            'The directory service has exhausted the pool of relative identifiers.';
    Win32ErrorCodes.ERROR_DS_INCORRECT_ROLE_OWNER:
        Win32ErrorCodeDescription := 'The requested operation could not be performed because the directory service is not the master for that type of operation.';
    Win32ErrorCodes.ERROR_DS_RIDMGR_INIT_ERROR:
        Win32ErrorCodeDescription := 'The directory service was unable to initialize the subsystem that allocates relative identifiers.';
    Win32ErrorCodes.ERROR_DS_OBJ_CLASS_VIOLATION:
        Win32ErrorCodeDescription := 'The requested operation did not satisfy one or more constraints associated with the class of the object.';
    Win32ErrorCodes.ERROR_DS_CANT_ON_NON_LEAF:
        Win32ErrorCodeDescription :=
            'The directory service can perform the requested operation only on a leaf object.';
    Win32ErrorCodes.ERROR_DS_CANT_ON_RDN:
        Win32ErrorCodeDescription := 'The directory service cannot perform the requested operation on the RDN attribute of an object.';
    Win32ErrorCodes.ERROR_DS_CANT_MOD_OBJ_CLASS:
        Win32ErrorCodeDescription :=
            'The directory service detected an attempt to modify the object class of an object.';
    Win32ErrorCodes.ERROR_DS_CROSS_DOM_MOVE_ERROR:
        Win32ErrorCodeDescription :=
            'The requested cross-domain move operation could not be performed.';
    Win32ErrorCodes.ERROR_DS_GC_NOT_AVAILABLE:
        Win32ErrorCodeDescription := 'Unable to contact the global catalog server.';
    Win32ErrorCodes.ERROR_SHARED_POLICY:
        Win32ErrorCodeDescription :=
            'The policy object is shared and can only be modified at the root.';
    Win32ErrorCodes.ERROR_POLICY_OBJECT_NOT_FOUND:
        Win32ErrorCodeDescription := 'The policy object does not exist.';
    Win32ErrorCodes.ERROR_POLICY_ONLY_IN_DS:
        Win32ErrorCodeDescription :=
            'The requested policy information is only in the directory service.';
    Win32ErrorCodes.ERROR_PROMOTION_ACTIVE:
        Win32ErrorCodeDescription := 'A domain controller promotion is currently active.';
    Win32ErrorCodes.ERROR_NO_PROMOTION_ACTIVE:
        Win32ErrorCodeDescription := 'A domain controller promotion is not currently active';
    Win32ErrorCodes.ERROR_DS_OPERATIONS_ERROR:
        Win32ErrorCodeDescription := 'An operations error occurred.';
    Win32ErrorCodes.ERROR_DS_PROTOCOL_ERROR:
        Win32ErrorCodeDescription := 'A protocol error occurred.';
    Win32ErrorCodes.ERROR_DS_TIMELIMIT_EXCEEDED:
        Win32ErrorCodeDescription := 'The time limit for this request was exceeded.';
    Win32ErrorCodes.ERROR_DS_SIZELIMIT_EXCEEDED:
        Win32ErrorCodeDescription := 'The size limit for this request was exceeded.';
    Win32ErrorCodes.ERROR_DS_ADMIN_LIMIT_EXCEEDED:
        Win32ErrorCodeDescription := 'The administrative limit for this request was exceeded.';
    Win32ErrorCodes.ERROR_DS_COMPARE_FALSE:
        Win32ErrorCodeDescription := 'The compare response was false.';
    Win32ErrorCodes.ERROR_DS_COMPARE_TRUE:
        Win32ErrorCodeDescription := 'The compare response was true.';
    Win32ErrorCodes.ERROR_DS_AUTH_METHOD_NOT_SUPPORTED:
        Win32ErrorCodeDescription :=
            'The requested authentication method is not supported by the server.';
    Win32ErrorCodes.ERROR_DS_STRONG_AUTH_REQUIRED:
        Win32ErrorCodeDescription :=
            'A more secure authentication method is required for this server.';
    Win32ErrorCodes.ERROR_DS_INAPPROPRIATE_AUTH:
        Win32ErrorCodeDescription := 'Inappropriate authentication.';
    Win32ErrorCodes.ERROR_DS_AUTH_UNKNOWN:
        Win32ErrorCodeDescription := 'The authentication mechanism is unknown.';
    Win32ErrorCodes.ERROR_DS_REFERRAL:
        Win32ErrorCodeDescription := 'A referral was returned from the server.';
    Win32ErrorCodes.ERROR_DS_UNAVAILABLE_CRIT_EXTENSION:
        Win32ErrorCodeDescription :=
            'The server does not support the requested critical extension.';
    Win32ErrorCodes.ERROR_DS_CONFIDENTIALITY_REQUIRED:
        Win32ErrorCodeDescription := 'This request requires a secure connection.';
    Win32ErrorCodes.ERROR_DS_INAPPROPRIATE_MATCHING:
        Win32ErrorCodeDescription := 'Inappropriate matching.';
    Win32ErrorCodes.ERROR_DS_CONSTRAINT_VIOLATION:
        Win32ErrorCodeDescription := 'A constraint violation occurred.';
    Win32ErrorCodes.ERROR_DS_NO_SUCH_OBJECT:
        Win32ErrorCodeDescription := 'There is no such object on the server.';
    Win32ErrorCodes.ERROR_DS_ALIAS_PROBLEM:
        Win32ErrorCodeDescription := 'There is an alias problem.';
    Win32ErrorCodes.ERROR_DS_INVALID_DN_SYNTAX:
        Win32ErrorCodeDescription := 'An invalid dn syntax has been specified.';
    Win32ErrorCodes.ERROR_DS_IS_LEAF:
        Win32ErrorCodeDescription := 'The object is a leaf object.';
    Win32ErrorCodes.ERROR_DS_ALIAS_DEREF_PROBLEM:
        Win32ErrorCodeDescription := 'There is an alias dereferencing problem.';
    Win32ErrorCodes.ERROR_DS_UNWILLING_TO_PERFORM:
        Win32ErrorCodeDescription := 'The server is unwilling to process the request.';
    Win32ErrorCodes.ERROR_DS_LOOP_DETECT:
        Win32ErrorCodeDescription := 'A loop has been detected.';
    Win32ErrorCodes.ERROR_DS_NAMING_VIOLATION:
        Win32ErrorCodeDescription := 'There is a naming violation.';
    Win32ErrorCodes.ERROR_DS_OBJECT_RESULTS_TOO_LARGE:
        Win32ErrorCodeDescription := 'The result set is too large.';
    Win32ErrorCodes.ERROR_DS_AFFECTS_MULTIPLE_DSAS:
        Win32ErrorCodeDescription := 'The operation affects multiple DSAs';
    Win32ErrorCodes.ERROR_DS_SERVER_DOWN:
        Win32ErrorCodeDescription := 'The server is not operational.';
    Win32ErrorCodes.ERROR_DS_LOCAL_ERROR:
        Win32ErrorCodeDescription := 'A local error has occurred.';
    Win32ErrorCodes.ERROR_DS_ENCODING_ERROR:
        Win32ErrorCodeDescription := 'An encoding error has occurred.';
    Win32ErrorCodes.ERROR_DS_DECODING_ERROR:
        Win32ErrorCodeDescription := 'A decoding error has occurred.';
    Win32ErrorCodes.ERROR_DS_FILTER_UNKNOWN:
        Win32ErrorCodeDescription := 'The search filter cannot be recognized.';
    Win32ErrorCodes.ERROR_DS_PARAM_ERROR:
        Win32ErrorCodeDescription := 'One or more parameters are illegal.';
    Win32ErrorCodes.ERROR_DS_NOT_SUPPORTED:
        Win32ErrorCodeDescription := 'The specified method is not supported.';
    Win32ErrorCodes.ERROR_DS_NO_RESULTS_RETURNED:
        Win32ErrorCodeDescription := 'No results were returned.';
    Win32ErrorCodes.ERROR_DS_CONTROL_NOT_FOUND:
        Win32ErrorCodeDescription := 'The specified control is not supported by the server.';
    Win32ErrorCodes.ERROR_DS_CLIENT_LOOP:
        Win32ErrorCodeDescription := 'A referral loop was detected by the client.';
    Win32ErrorCodes.ERROR_DS_REFERRAL_LIMIT_EXCEEDED:
        Win32ErrorCodeDescription := 'The preset referral limit was exceeded.';
    Win32ErrorCodes.ERROR_DS_SORT_CONTROL_MISSING:
        Win32ErrorCodeDescription := 'The search requires a SORT control.';
    Win32ErrorCodes.ERROR_DS_OFFSET_RANGE_ERROR:
        Win32ErrorCodeDescription := 'The search results exceed the offset range specified.';
    Win32ErrorCodes.ERROR_DS_ROOT_MUST_BE_NC:
        Win32ErrorCodeDescription := 'The root object must be the head of a naming context. The root object cannot have an instantiated parent.';
    Win32ErrorCodes.ERROR_DS_ADD_REPLICA_INHIBITED:
        Win32ErrorCodeDescription := 'The add replica operation cannot be performed. The naming context must be writable in order to create the replica.';
    Win32ErrorCodes.ERROR_DS_ATT_NOT_DEF_IN_SCHEMA:
        Win32ErrorCodeDescription :=
            'A reference to an attribute that is not defined in the schema occurred.';
    Win32ErrorCodes.ERROR_DS_MAX_OBJ_SIZE_EXCEEDED:
        Win32ErrorCodeDescription := 'The maximum size of an object has been exceeded.';
    Win32ErrorCodes.ERROR_DS_OBJ_STRING_NAME_EXISTS:
        Win32ErrorCodeDescription :=
            'An attempt was made to add an object to the directory with a name that is already in use.';
    Win32ErrorCodes.ERROR_DS_NO_RDN_DEFINED_IN_SCHEMA:
        Win32ErrorCodeDescription := 'An attempt was made to add an object of a class that does not have an RDN defined in the schema.';
    Win32ErrorCodes.ERROR_DS_RDN_DOESNT_MATCH_SCHEMA:
        Win32ErrorCodeDescription := 'An attempt was made to add an object using an RDN that is not the RDN defined in the schema.';
    Win32ErrorCodes.ERROR_DS_NO_REQUESTED_ATTS_FOUND:
        Win32ErrorCodeDescription := 'None of the requested attributes were found on the objects.';
    Win32ErrorCodes.ERROR_DS_USER_BUFFER_TO_SMALL:
        Win32ErrorCodeDescription := 'The user buffer is too small.';
    Win32ErrorCodes.ERROR_DS_ATT_IS_NOT_ON_OBJ:
        Win32ErrorCodeDescription :=
            'The attribute specified in the operation is not present on the object.';
    Win32ErrorCodes.ERROR_DS_ILLEGAL_MOD_OPERATION:
        Win32ErrorCodeDescription :=
            'Illegal modify operation. Some aspect of the modification is not permitted.';
    Win32ErrorCodes.ERROR_DS_OBJ_TOO_LARGE:
        Win32ErrorCodeDescription := 'The specified object is too large.';
    Win32ErrorCodes.ERROR_DS_BAD_INSTANCE_TYPE:
        Win32ErrorCodeDescription := 'The specified instance type is not valid.';
    Win32ErrorCodes.ERROR_DS_MASTERDSA_REQUIRED:
        Win32ErrorCodeDescription := 'The operation must be performed at a master DSA.';
    Win32ErrorCodes.ERROR_DS_OBJECT_CLASS_REQUIRED:
        Win32ErrorCodeDescription := 'The object class attribute must be specified.';
    Win32ErrorCodes.ERROR_DS_MISSING_REQUIRED_ATT:
        Win32ErrorCodeDescription := 'A required attribute is missing.';
    Win32ErrorCodes.ERROR_DS_ATT_NOT_DEF_FOR_CLASS:
        Win32ErrorCodeDescription := 'An attempt was made to modify an object to include an attribute that is not legal for its class';
    Win32ErrorCodes.ERROR_DS_ATT_ALREADY_EXISTS:
        Win32ErrorCodeDescription := 'The specified attribute is already present on the object.';
    Win32ErrorCodes.ERROR_DS_CANT_ADD_ATT_VALUES:
        Win32ErrorCodeDescription := 'The specified attribute is not present, or has no values.';
    Win32ErrorCodes.ERROR_DS_SINGLE_VALUE_CONSTRAINT:
        Win32ErrorCodeDescription :=
            'Multiple values were specified for an attribute that can have only one value.';
    Win32ErrorCodes.ERROR_DS_RANGE_CONSTRAINT:
        Win32ErrorCodeDescription :=
            'A value for the attribute was not in the acceptable range of values.';
    Win32ErrorCodes.ERROR_DS_ATT_VAL_ALREADY_EXISTS:
        Win32ErrorCodeDescription := 'The specified value already exists.';
    Win32ErrorCodes.ERROR_DS_CANT_REM_MISSING_ATT:
        Win32ErrorCodeDescription :=
            'The attribute cannot be removed because it is not present on the object.';
    Win32ErrorCodes.ERROR_DS_CANT_REM_MISSING_ATT_VAL:
        Win32ErrorCodeDescription :=
            'The attribute value cannot be removed because it is not present on the object.';
    Win32ErrorCodes.ERROR_DS_ROOT_CANT_BE_SUBREF:
        Win32ErrorCodeDescription := 'The specified root object cannot be a subref.';
    Win32ErrorCodes.ERROR_DS_NO_CHAINING:
        Win32ErrorCodeDescription := 'Chaining is not permitted.';
    Win32ErrorCodes.ERROR_DS_NO_CHAINED_EVAL:
        Win32ErrorCodeDescription := 'Chained evaluation is not permitted.';
    Win32ErrorCodes.ERROR_DS_NO_PARENT_OBJECT:
        Win32ErrorCodeDescription := 'The operation could not be performed because the objects parent is either uninstantiated or deleted.';
    Win32ErrorCodes.ERROR_DS_PARENT_IS_AN_ALIAS:
        Win32ErrorCodeDescription :=
            'Having a parent that is an alias is not permitted. Aliases are leaf objects.';
    Win32ErrorCodes.ERROR_DS_CANT_MIX_MASTER_AND_REPS:
        Win32ErrorCodeDescription :=
            'The object and parent must be of the same type, either both masters or both replicas.';
    Win32ErrorCodes.ERROR_DS_CHILDREN_EXIST:
        Win32ErrorCodeDescription := 'The operation cannot be performed because child objects exist. This operation can only be performed on a leaf object.';
    Win32ErrorCodes.ERROR_DS_OBJ_NOT_FOUND:
        Win32ErrorCodeDescription := 'Directory object not found.';
    Win32ErrorCodes.ERROR_DS_ALIASED_OBJ_MISSING:
        Win32ErrorCodeDescription := 'The aliased object is missing.';
    Win32ErrorCodes.ERROR_DS_BAD_NAME_SYNTAX:
        Win32ErrorCodeDescription := 'The object name has bad syntax.';
    Win32ErrorCodes.ERROR_DS_ALIAS_POINTS_TO_ALIAS:
        Win32ErrorCodeDescription := 'It is not permitted for an alias to refer to another alias.';
    Win32ErrorCodes.ERROR_DS_CANT_DEREF_ALIAS:
        Win32ErrorCodeDescription := 'The alias cannot be dereferenced.';
    Win32ErrorCodes.ERROR_DS_OUT_OF_SCOPE:
        Win32ErrorCodeDescription := 'The operation is out of scope.';
    Win32ErrorCodes.ERROR_DS_OBJECT_BEING_REMOVED:
        Win32ErrorCodeDescription :=
            'The operation cannot continue because the object is in the process of being removed.';
    Win32ErrorCodes.ERROR_DS_CANT_DELETE_DSA_OBJ:
        Win32ErrorCodeDescription := 'The DSA object cannot be deleted.';
    Win32ErrorCodes.ERROR_DS_GENERIC_ERROR:
        Win32ErrorCodeDescription := 'A directory service error has occurred.';
    Win32ErrorCodes.ERROR_DS_DSA_MUST_BE_INT_MASTER:
        Win32ErrorCodeDescription :=
            'The operation can only be performed on an internal master DSA object.';
    Win32ErrorCodes.ERROR_DS_CLASS_NOT_DSA:
        Win32ErrorCodeDescription := 'The object must be of class DSA.';
    Win32ErrorCodes.ERROR_DS_INSUFF_ACCESS_RIGHTS:
        Win32ErrorCodeDescription := 'Insufficient access rights to perform the operation.';
    Win32ErrorCodes.ERROR_DS_ILLEGAL_SUPERIOR:
        Win32ErrorCodeDescription :=
            'The object cannot be added because the parent is not on the list of possible superiors.';
    Win32ErrorCodes.ERROR_DS_ATTRIBUTE_OWNED_BY_SAM:
        Win32ErrorCodeDescription := 'Access to the attribute is not permitted because the attribute is owned by the Security Accounts Manager (SAM).';
    Win32ErrorCodes.ERROR_DS_NAME_TOO_MANY_PARTS:
        Win32ErrorCodeDescription := 'The name has too many parts.';
    Win32ErrorCodes.ERROR_DS_NAME_TOO_LONG:
        Win32ErrorCodeDescription := 'The name is too long.';
    Win32ErrorCodes.ERROR_DS_NAME_VALUE_TOO_LONG:
        Win32ErrorCodeDescription := 'The name value is too long.';
    Win32ErrorCodes.ERROR_DS_NAME_UNPARSEABLE:
        Win32ErrorCodeDescription := 'The directory service encountered an error parsing a name.';
    Win32ErrorCodes.ERROR_DS_NAME_TYPE_UNKNOWN:
        Win32ErrorCodeDescription :=
            'The directory service cannot get the attribute type for a name.';
    Win32ErrorCodes.ERROR_DS_NOT_AN_OBJECT:
        Win32ErrorCodeDescription :=
            'The name does not identify an object; the name identifies a phantom.';
    Win32ErrorCodes.ERROR_DS_SEC_DESC_TOO_SHORT:
        Win32ErrorCodeDescription := 'The security descriptor is too short.';
    Win32ErrorCodes.ERROR_DS_SEC_DESC_INVALID:
        Win32ErrorCodeDescription := 'The security descriptor is invalid.';
    Win32ErrorCodes.ERROR_DS_NO_DELETED_NAME:
        Win32ErrorCodeDescription := 'Failed to create name for deleted object.';
    Win32ErrorCodes.ERROR_DS_SUBREF_MUST_HAVE_PARENT:
        Win32ErrorCodeDescription := 'The parent of a new subref must exist.';
    Win32ErrorCodes.ERROR_DS_NCNAME_MUST_BE_NC:
        Win32ErrorCodeDescription := 'The object must be a naming context.';
    Win32ErrorCodes.ERROR_DS_CANT_ADD_SYSTEM_ONLY:
        Win32ErrorCodeDescription :=
            'It is not permitted to add an attribute which is owned by the system.';
    Win32ErrorCodes.ERROR_DS_CLASS_MUST_BE_CONCRETE:
        Win32ErrorCodeDescription :=
            'The class of the object must be structural; you cannot instantiate an abstract class.';
    Win32ErrorCodes.ERROR_DS_INVALID_DMD:
        Win32ErrorCodeDescription := 'The schema object could not be found.';
    Win32ErrorCodes.ERROR_DS_OBJ_GUID_EXISTS:
        Win32ErrorCodeDescription :=
            'A local object with this GUID (dead or alive) already exists.';
    Win32ErrorCodes.ERROR_DS_NOT_ON_BACKLINK:
        Win32ErrorCodeDescription := 'The operation cannot be performed on a back link.';
    Win32ErrorCodes.ERROR_DS_NO_CROSSREF_FOR_NC:
        Win32ErrorCodeDescription :=
            'The cross reference for the specified naming context could not be found.';
    Win32ErrorCodes.ERROR_DS_SHUTTING_DOWN:
        Win32ErrorCodeDescription :=
            'The operation could not be performed because the directory service is shutting down.';
    Win32ErrorCodes.ERROR_DS_UNKNOWN_OPERATION:
        Win32ErrorCodeDescription := 'The directory service request is invalid.';
    Win32ErrorCodes.ERROR_DS_INVALID_ROLE_OWNER:
        Win32ErrorCodeDescription := 'The role owner attribute could not be read.';
    Win32ErrorCodes.ERROR_DS_COULDNT_CONTACT_FSMO:
        Win32ErrorCodeDescription :=
            'The requested FSMO operation failed. The current FSMO holder could not be reached.';
    Win32ErrorCodes.ERROR_DS_CROSS_NC_DN_RENAME:
        Win32ErrorCodeDescription :=
            'Modification of a DN across a naming context is not permitted.';
    Win32ErrorCodes.ERROR_DS_CANT_MOD_SYSTEM_ONLY:
        Win32ErrorCodeDescription :=
            'The attribute cannot be modified because it is owned by the system.';
    Win32ErrorCodes.ERROR_DS_REPLICATOR_ONLY:
        Win32ErrorCodeDescription := 'Only the replicator can perform this function.';
    Win32ErrorCodes.ERROR_DS_OBJ_CLASS_NOT_DEFINED:
        Win32ErrorCodeDescription := 'The specified class is not defined.';
    Win32ErrorCodes.ERROR_DS_OBJ_CLASS_NOT_SUBCLASS:
        Win32ErrorCodeDescription := 'The specified class is not a subclass.';
    Win32ErrorCodes.ERROR_DS_NAME_REFERENCE_INVALID:
        Win32ErrorCodeDescription := 'The name reference is invalid.';
    Win32ErrorCodes.ERROR_DS_CROSS_REF_EXISTS:
        Win32ErrorCodeDescription := 'A cross reference already exists.';
    Win32ErrorCodes.ERROR_DS_CANT_DEL_MASTER_CROSSREF:
        Win32ErrorCodeDescription := 'It is not permitted to delete a master cross reference.';
    Win32ErrorCodes.ERROR_DS_SUBTREE_NOTIFY_NOT_NC_HEAD:
        Win32ErrorCodeDescription := 'Subtree notifications are only supported on NC heads.';
    Win32ErrorCodes.ERROR_DS_NOTIFY_FILTER_TOO_COMPLEX:
        Win32ErrorCodeDescription := 'Notification filter is too complex.';
    Win32ErrorCodes.ERROR_DS_DUP_RDN:
        Win32ErrorCodeDescription := 'Schema update failed: duplicate RDN.';
    Win32ErrorCodes.ERROR_DS_DUP_OID:
        Win32ErrorCodeDescription := 'Schema update failed: duplicate OID';
    Win32ErrorCodes.ERROR_DS_DUP_MAPI_ID:
        Win32ErrorCodeDescription := 'Schema update failed: duplicate MAPI identifier.';
    Win32ErrorCodes.ERROR_DS_DUP_SCHEMA_ID_GUID:
        Win32ErrorCodeDescription := 'Schema update failed: duplicate schema-id GUID.';
    Win32ErrorCodes.ERROR_DS_DUP_LDAP_DISPLAY_NAME:
        Win32ErrorCodeDescription := 'Schema update failed: duplicate LDAP display name.';
    Win32ErrorCodes.ERROR_DS_SEMANTIC_ATT_TEST:
        Win32ErrorCodeDescription := 'Schema update failed: range-lower less than range upper';
    Win32ErrorCodes.ERROR_DS_SYNTAX_MISMATCH:
        Win32ErrorCodeDescription := 'Schema update failed: syntax mismatch';
    Win32ErrorCodes.ERROR_DS_EXISTS_IN_MUST_HAVE:
        Win32ErrorCodeDescription := 'Schema deletion failed: attribute is used in must-contain';
    Win32ErrorCodes.ERROR_DS_EXISTS_IN_MAY_HAVE:
        Win32ErrorCodeDescription := 'Schema deletion failed: attribute is used in may-contain';
    Win32ErrorCodes.ERROR_DS_NONEXISTENT_MAY_HAVE:
        Win32ErrorCodeDescription :=
            'Schema update failed: attribute in may-contain does not exist';
    Win32ErrorCodes.ERROR_DS_NONEXISTENT_MUST_HAVE:
        Win32ErrorCodeDescription :=
            'Schema update failed: attribute in must-contain does not exist';
    Win32ErrorCodes.ERROR_DS_AUX_CLS_TEST_FAIL:
        Win32ErrorCodeDescription :=
            'Schema update failed: class in aux-class list does not exist or is not an auxiliary class';
    Win32ErrorCodes.ERROR_DS_NONEXISTENT_POSS_SUP:
        Win32ErrorCodeDescription :=
            'Schema update failed: class in poss-superiors does not exist';
    Win32ErrorCodes.ERROR_DS_SUB_CLS_TEST_FAIL:
        Win32ErrorCodeDescription := 'Schema update failed: class in subclassof list does not exist or does not satisfy hierarchy rules';
    Win32ErrorCodes.ERROR_DS_BAD_RDN_ATT_ID_SYNTAX:
        Win32ErrorCodeDescription := 'Schema update failed: Rdn-Att-Id has wrong syntax';
    Win32ErrorCodes.ERROR_DS_EXISTS_IN_AUX_CLS:
        Win32ErrorCodeDescription := 'Schema deletion failed: class is used as auxiliary class';
    Win32ErrorCodes.ERROR_DS_EXISTS_IN_SUB_CLS:
        Win32ErrorCodeDescription := 'Schema deletion failed: class is used as sub class';
    Win32ErrorCodes.ERROR_DS_EXISTS_IN_POSS_SUP:
        Win32ErrorCodeDescription := 'Schema deletion failed: class is used as poss superior';
    Win32ErrorCodes.ERROR_DS_RECALCSCHEMA_FAILED:
        Win32ErrorCodeDescription := 'Schema update failed in recalculating validation cache.';
    Win32ErrorCodes.ERROR_DS_TREE_DELETE_NOT_FINISHED:
        Win32ErrorCodeDescription := 'The tree deletion is not finished.';
    Win32ErrorCodes.ERROR_DS_CANT_DELETE:
        Win32ErrorCodeDescription := 'The requested delete operation could not be performed.';
    Win32ErrorCodes.ERROR_DS_ATT_SCHEMA_REQ_ID:
        Win32ErrorCodeDescription :=
            'Cannot read the governs class identifier for the schema record.';
    Win32ErrorCodes.ERROR_DS_BAD_ATT_SCHEMA_SYNTAX:
        Win32ErrorCodeDescription := 'The attribute schema has bad syntax.';
    Win32ErrorCodes.ERROR_DS_CANT_CACHE_ATT:
        Win32ErrorCodeDescription := 'The attribute could not be cached.';
    Win32ErrorCodes.ERROR_DS_CANT_CACHE_CLASS:
        Win32ErrorCodeDescription := 'The class could not be cached.';
    Win32ErrorCodes.ERROR_DS_CANT_REMOVE_ATT_CACHE:
        Win32ErrorCodeDescription := 'The attribute could not be removed from the cache.';
    Win32ErrorCodes.ERROR_DS_CANT_REMOVE_CLASS_CACHE:
        Win32ErrorCodeDescription := 'The class could not be removed from the cache.';
    Win32ErrorCodes.ERROR_DS_CANT_RETRIEVE_DN:
        Win32ErrorCodeDescription := 'The distinguished name attribute could not be read.';
    Win32ErrorCodes.ERROR_DS_MISSING_SUPREF:
        Win32ErrorCodeDescription := 'A required subref is missing.';
    Win32ErrorCodes.ERROR_DS_CANT_RETRIEVE_INSTANCE:
        Win32ErrorCodeDescription := 'The instance type attribute could not be retrieved.';
    Win32ErrorCodes.ERROR_DS_CODE_INCONSISTENCY:
        Win32ErrorCodeDescription := 'An internal error has occurred.';
    Win32ErrorCodes.ERROR_DS_DATABASE_ERROR:
        Win32ErrorCodeDescription := 'A database error has occurred.';
    Win32ErrorCodes.ERROR_DS_GOVERNSID_MISSING:
        Win32ErrorCodeDescription := 'The attribute GOVERNSID is missing.';
    Win32ErrorCodes.ERROR_DS_MISSING_EXPECTED_ATT:
        Win32ErrorCodeDescription := 'An expected attribute is missing.';
    Win32ErrorCodes.ERROR_DS_NCNAME_MISSING_CR_REF:
        Win32ErrorCodeDescription := 'The specified naming context is missing a cross reference.';
    Win32ErrorCodes.ERROR_DS_SECURITY_CHECKING_ERROR:
        Win32ErrorCodeDescription := 'A security checking error has occurred.';
    Win32ErrorCodes.ERROR_DS_SCHEMA_NOT_LOADED:
        Win32ErrorCodeDescription := 'The schema is not loaded.';
    Win32ErrorCodes.ERROR_DS_SCHEMA_ALLOC_FAILED:
        Win32ErrorCodeDescription :=
            'Schema allocation failed. Please check if the machine is running low on memory.';
    Win32ErrorCodes.ERROR_DS_ATT_SCHEMA_REQ_SYNTAX:
        Win32ErrorCodeDescription :=
            'Failed to obtain the required syntax for the attribute schema.';
    Win32ErrorCodes.ERROR_DS_GCVERIFY_ERROR:
        Win32ErrorCodeDescription := 'The global catalog verification failed. The global catalog is not available or does not support the operation. Some part of the directory is currently not available.';
    Win32ErrorCodes.ERROR_DS_DRA_SCHEMA_MISMATCH:
        Win32ErrorCodeDescription := 'The replication operation failed because of a schema mismatch between the servers involved.';
    Win32ErrorCodes.ERROR_DS_CANT_FIND_DSA_OBJ:
        Win32ErrorCodeDescription := 'The DSA object could not be found.';
    Win32ErrorCodes.ERROR_DS_CANT_FIND_EXPECTED_NC:
        Win32ErrorCodeDescription := 'The naming context could not be found.';
    Win32ErrorCodes.ERROR_DS_CANT_FIND_NC_IN_CACHE:
        Win32ErrorCodeDescription := 'The naming context could not be found in the cache.';
    Win32ErrorCodes.ERROR_DS_CANT_RETRIEVE_CHILD:
        Win32ErrorCodeDescription := 'The child object could not be retrieved.';
    Win32ErrorCodes.ERROR_DS_SECURITY_ILLEGAL_MODIFY:
        Win32ErrorCodeDescription := 'The modification was not permitted for security reasons.';
    Win32ErrorCodes.ERROR_DS_CANT_REPLACE_HIDDEN_REC:
        Win32ErrorCodeDescription := 'The operation cannot replace the hidden record.';
    Win32ErrorCodes.ERROR_DS_BAD_HIERARCHY_FILE:
        Win32ErrorCodeDescription := 'The hierarchy file is invalid.';
    Win32ErrorCodes.ERROR_DS_BUILD_HIERARCHY_TABLE_FAILED:
        Win32ErrorCodeDescription := 'The attempt to build the hierarchy table failed.';
    Win32ErrorCodes.ERROR_DS_CONFIG_PARAM_MISSING:
        Win32ErrorCodeDescription :=
            'The directory configuration parameter is missing from the registry.';
    Win32ErrorCodes.ERROR_DS_COUNTING_AB_INDICES_FAILED:
        Win32ErrorCodeDescription := 'The attempt to count the address book indices failed.';
    Win32ErrorCodes.ERROR_DS_HIERARCHY_TABLE_MALLOC_FAILED:
        Win32ErrorCodeDescription := 'The allocation of the hierarchy table failed.';
    Win32ErrorCodes.ERROR_DS_INTERNAL_FAILURE:
        Win32ErrorCodeDescription := 'The directory service encountered an internal failure.';
    Win32ErrorCodes.ERROR_DS_UNKNOWN_ERROR:
        Win32ErrorCodeDescription := 'The directory service encountered an unknown failure.';
    Win32ErrorCodes.ERROR_DS_ROOT_REQUIRES_CLASS_TOP:
        Win32ErrorCodeDescription := 'A root object requires a class of top.';
    Win32ErrorCodes.ERROR_DS_REFUSING_FSMO_ROLES:
        Win32ErrorCodeDescription := 'This directory server is shutting down, and cannot take ownership of new floating single-master operation roles.';
    Win32ErrorCodes.ERROR_DS_MISSING_FSMO_SETTINGS:
        Win32ErrorCodeDescription := 'The directory service is missing mandatory configuration information, and is unable to determine the ownership of floating single-master operation roles.';
    Win32ErrorCodes.ERROR_DS_UNABLE_TO_SURRENDER_ROLES:
        Win32ErrorCodeDescription := 'The directory service was unable to transfer ownership of one or more floating single-master operation roles to other servers.';
    Win32ErrorCodes.ERROR_DS_DRA_GENERIC:
        Win32ErrorCodeDescription := 'The replication operation failed.';
    Win32ErrorCodes.ERROR_DS_DRA_INVALID_PARAMETER:
        Win32ErrorCodeDescription :=
            'An invalid parameter was specified for this replication operation.';
    Win32ErrorCodes.ERROR_DS_DRA_BUSY:
        Win32ErrorCodeDescription :=
            'The directory service is too busy to complete the replication operation at this time.';
    Win32ErrorCodes.ERROR_DS_DRA_BAD_DN:
        Win32ErrorCodeDescription :=
            'The distinguished name specified for this replication operation is invalid.';
    Win32ErrorCodes.ERROR_DS_DRA_BAD_NC:
        Win32ErrorCodeDescription :=
            'The naming context specified for this replication operation is invalid.';
    Win32ErrorCodes.ERROR_DS_DRA_DN_EXISTS:
        Win32ErrorCodeDescription :=
            'The distinguished name specified for this replication operation already exists.';
    Win32ErrorCodes.ERROR_DS_DRA_INTERNAL_ERROR:
        Win32ErrorCodeDescription := 'The replication system encountered an internal error.';
    Win32ErrorCodes.ERROR_DS_DRA_INCONSISTENT_DIT:
        Win32ErrorCodeDescription :=
            'The replication operation encountered a database inconsistency.';
    Win32ErrorCodes.ERROR_DS_DRA_CONNECTION_FAILED:
        Win32ErrorCodeDescription :=
            'The server specified for this replication operation could not be contacted.';
    Win32ErrorCodes.ERROR_DS_DRA_BAD_INSTANCE_TYPE:
        Win32ErrorCodeDescription :=
            'The replication operation encountered an object with an invalid instance type.';
    Win32ErrorCodes.ERROR_DS_DRA_OUT_OF_MEM:
        Win32ErrorCodeDescription := 'The replication operation failed to allocate memory.';
    Win32ErrorCodes.ERROR_DS_DRA_MAIL_PROBLEM:
        Win32ErrorCodeDescription :=
            'The replication operation encountered an error with the mail system.';
    Win32ErrorCodes.ERROR_DS_DRA_REF_ALREADY_EXISTS:
        Win32ErrorCodeDescription :=
            'The replication reference information for the target server already exists.';
    Win32ErrorCodes.ERROR_DS_DRA_REF_NOT_FOUND:
        Win32ErrorCodeDescription :=
            'The replication reference information for the target server does not exist.';
    Win32ErrorCodes.ERROR_DS_DRA_OBJ_IS_REP_SOURCE:
        Win32ErrorCodeDescription :=
            'The naming context cannot be removed because it is replicated to another server.';
    Win32ErrorCodes.ERROR_DS_DRA_DB_ERROR:
        Win32ErrorCodeDescription := 'The replication operation encountered a database error.';
    Win32ErrorCodes.ERROR_DS_DRA_NO_REPLICA:
        Win32ErrorCodeDescription := 'The naming context is in the process of being removed or is not replicated from the specified server.';
    Win32ErrorCodes.ERROR_DS_DRA_ACCESS_DENIED:
        Win32ErrorCodeDescription := 'Replication access was denied.';
    Win32ErrorCodes.ERROR_DS_DRA_NOT_SUPPORTED:
        Win32ErrorCodeDescription :=
            'The requested operation is not supported by this version of the directory service.';
    Win32ErrorCodes.ERROR_DS_DRA_RPC_CANCELLED:
        Win32ErrorCodeDescription := 'The replication remote procedure call was cancelled.';
    Win32ErrorCodes.ERROR_DS_DRA_SOURCE_DISABLED:
        Win32ErrorCodeDescription :=
            'The source server is currently rejecting replication requests.';
    Win32ErrorCodes.ERROR_DS_DRA_SINK_DISABLED:
        Win32ErrorCodeDescription :=
            'The destination server is currently rejecting replication requests.';
    Win32ErrorCodes.ERROR_DS_DRA_NAME_COLLISION:
        Win32ErrorCodeDescription :=
            'The replication operation failed due to a collision of object names.';
    Win32ErrorCodes.ERROR_DS_DRA_SOURCE_REINSTALLED:
        Win32ErrorCodeDescription := 'The replication source has been reinstalled.';
    Win32ErrorCodes.ERROR_DS_DRA_MISSING_PARENT:
        Win32ErrorCodeDescription :=
            'The replication operation failed because a required parent object is missing.';
    Win32ErrorCodes.ERROR_DS_DRA_PREEMPTED:
        Win32ErrorCodeDescription := 'The replication operation was preempted.';
    Win32ErrorCodes.ERROR_DS_DRA_ABANDON_SYNC:
        Win32ErrorCodeDescription :=
            'The replication synchronization attempt was abandoned because of a lack of updates.';
    Win32ErrorCodes.ERROR_DS_DRA_SHUTDOWN:
        Win32ErrorCodeDescription :=
            'The replication operation was terminated because the system is shutting down.';
    Win32ErrorCodes.ERROR_DS_DRA_INCOMPATIBLE_PARTIAL_SET:
        Win32ErrorCodeDescription := 'The replication synchronization attempt failed as the destination partial attribute set is not a subset of source partial attribute set.';
    Win32ErrorCodes.ERROR_DS_DRA_SOURCE_IS_PARTIAL_REPLICA:
        Win32ErrorCodeDescription := 'The replication synchronization attempt failed because a master replica attempted to sync from a partial replica.';
    Win32ErrorCodes.ERROR_DS_DRA_EXTN_CONNECTION_FAILED:
        Win32ErrorCodeDescription := 'The server specified for this replication operation was contacted, but that server was unable to contact an additional server needed to complete the operation.';
    Win32ErrorCodes.ERROR_DS_INSTALL_SCHEMA_MISMATCH:
        Win32ErrorCodeDescription := 'The version of the Active Directory (AD) schema of the source forest is not compatible with the version of AD on this computer. Upgrade the operating system on a domain controller in the source forest before it can be added as a controller to that forest.';
    Win32ErrorCodes.ERROR_DS_DUP_LINK_ID:
        Win32ErrorCodeDescription :=
            'Schema update failed: An attribute with the same link identifier already exists.';
    Win32ErrorCodes.ERROR_DS_NAME_ERROR_RESOLVING:
        Win32ErrorCodeDescription := 'Name translation: Generic processing error.';
    Win32ErrorCodes.ERROR_DS_NAME_ERROR_NOT_FOUND:
        Win32ErrorCodeDescription :=
            'Name translation: Could not find the name or insufficient right to see name.';
    Win32ErrorCodes.ERROR_DS_NAME_ERROR_NOT_UNIQUE:
        Win32ErrorCodeDescription :=
            'Name translation: Input name mapped to more than one output name.';
    Win32ErrorCodes.ERROR_DS_NAME_ERROR_NO_MAPPING:
        Win32ErrorCodeDescription :=
            'Name translation: Input name found, but not the associated output format.';
    Win32ErrorCodes.ERROR_DS_NAME_ERROR_DOMAIN_ONLY:
        Win32ErrorCodeDescription :=
            'Name translation: Unable to resolve completely, only the domain was found.';
    Win32ErrorCodes.ERROR_DS_NAME_ERROR_NO_SYNTACTICAL_MAPPING:
        Win32ErrorCodeDescription := 'Name translation: Unable to perform purely syntactical mapping at the client without going out to the wire.';
    Win32ErrorCodes.ERROR_DS_CONSTRUCTED_ATT_MOD:
        Win32ErrorCodeDescription := 'Modification of a constructed att is not allowed.';
    Win32ErrorCodes.ERROR_DS_WRONG_OM_OBJ_CLASS:
        Win32ErrorCodeDescription :=
            'The OM-Object-Class specified is incorrect for an attribute with the specified syntax.';
    Win32ErrorCodes.ERROR_DS_DRA_REPL_PENDING:
        Win32ErrorCodeDescription := 'The replication request has been posted; waiting for reply.';
    Win32ErrorCodes.ERROR_DS_DS_REQUIRED:
        Win32ErrorCodeDescription :=
            'The requested operation requires a directory service, and none was available.';
    Win32ErrorCodes.ERROR_DS_INVALID_LDAP_DISPLAY_NAME:
        Win32ErrorCodeDescription :=
            'The LDAP display name of the class or attribute contains non-ASCII characters.';
    Win32ErrorCodes.ERROR_DS_NON_BASE_SEARCH:
        Win32ErrorCodeDescription :=
            'The requested search operation is only supported for base searches.';
    Win32ErrorCodes.ERROR_DS_CANT_RETRIEVE_ATTS:
        Win32ErrorCodeDescription := 'The search failed to retrieve attributes from the database.';
    Win32ErrorCodes.ERROR_DS_BACKLINK_WITHOUT_LINK:
        Win32ErrorCodeDescription := 'The schema update operation tried to add a backward link attribute that has no corresponding forward link.';
    Win32ErrorCodes.ERROR_DS_EPOCH_MISMATCH:
        Win32ErrorCodeDescription := 'Source and destination of a cross domain move do not agree on the objects epoch number. Either source or destination does not have the latest version of the object.';
    Win32ErrorCodes.ERROR_DS_SRC_NAME_MISMATCH:
        Win32ErrorCodeDescription := 'Source and destination of a cross domain move do not agree on the objects current name. Either source or destination does not have the latest version of the object.';
    Win32ErrorCodes.ERROR_DS_SRC_AND_DST_NC_IDENTICAL:
        Win32ErrorCodeDescription := 'Source and destination of a cross domain move operation are identical. Caller should use local move operation instead of cross domain move operation.';
    Win32ErrorCodes.ERROR_DS_DST_NC_MISMATCH:
        Win32ErrorCodeDescription := 'Source and destination for a cross domain move are not in agreement on the naming contexts in the forest. Either source or destination does not have the latest version of the Partitions container.';
    Win32ErrorCodes.ERROR_DS_NOT_AUTHORITIVE_FOR_DST_NC:
        Win32ErrorCodeDescription := 'Destination of a cross domain move is not authoritative for the destination naming context.';
    Win32ErrorCodes.ERROR_DS_SRC_GUID_MISMATCH:
        Win32ErrorCodeDescription := 'Source and destination of a cross domain move do not agree on the identity of the source object. Either source or destination does not have the latest version of the source object.';
    Win32ErrorCodes.ERROR_DS_CANT_MOVE_DELETED_OBJECT:
        Win32ErrorCodeDescription := 'Object being moved across domains is already known to be deleted by the destination server. The source server does not have the latest version of the source object.';
    Win32ErrorCodes.ERROR_DS_PDC_OPERATION_IN_PROGRESS:
        Win32ErrorCodeDescription :=
            'Another operation which requires exclusive access to the PDC PSMO is already in progress.';
    Win32ErrorCodes.ERROR_DS_CROSS_DOMAIN_CLEANUP_REQD:
        Win32ErrorCodeDescription := 'A cross domain move operation failed such that the two versions of the moved object exist - one each in the source and destination domains. The destination object needs to be removed to restore the system to a consistent state.';
    Win32ErrorCodes.ERROR_DS_ILLEGAL_XDOM_MOVE_OPERATION:
        Win32ErrorCodeDescription := 'This object may not be moved across domain boundaries either because cross domain moves for this class are disallowed, or the object has some special characteristics, eg: trust account or restricted RID, which prevent its move.';
    Win32ErrorCodes.ERROR_DS_CANT_WITH_ACCT_GROUP_MEMBERSHPS:
        Win32ErrorCodeDescription := 'Cant move objects with memberships across domain boundaries as once moved, this would violate the membership conditions of the account group. Remove the object from any account group memberships and retry.';
    Win32ErrorCodes.ERROR_DS_NC_MUST_HAVE_NC_PARENT:
        Win32ErrorCodeDescription := 'A naming context head must be the immediate child of another naming context head, not of an interior node.';
    Win32ErrorCodes.ERROR_DS_CR_IMPOSSIBLE_TO_VALIDATE:
        Win32ErrorCodeDescription := 'The directory cant validate the proposed naming context name because it doesnt hold a replica of the naming context above the proposed naming context.';
    Win32ErrorCodes.ERROR_DS_DST_DOMAIN_NOT_NATIVE:
        Win32ErrorCodeDescription := 'Destination domain must be in native mode.';
    Win32ErrorCodes.ERROR_DS_MISSING_INFRASTRUCTURE_CONTAINER:
        Win32ErrorCodeDescription := 'The operation can not be performed because the server does not have an infrastructure container in the domain of interest.';
    Win32ErrorCodes.ERROR_DS_CANT_MOVE_ACCOUNT_GROUP:
        Win32ErrorCodeDescription :=
            'Cross-domain move of non-empty account groups is not allowed.';
    Win32ErrorCodes.ERROR_DS_CANT_MOVE_RESOURCE_GROUP:
        Win32ErrorCodeDescription :=
            'Cross-domain move of non-empty resource groups is not allowed.';
    Win32ErrorCodes.ERROR_DS_INVALID_SEARCH_FLAG:
        Win32ErrorCodeDescription := 'The search flags for the attribute are invalid. The ANR bit is valid only on attributes of Unicode or Teletex strings.';
    Win32ErrorCodes.ERROR_DS_NO_TREE_DELETE_ABOVE_NC:
        Win32ErrorCodeDescription := 'Tree deletions starting at an object which has an NC head as a descendant are not allowed.';
    Win32ErrorCodes.ERROR_DS_COULDNT_LOCK_TREE_FOR_DELETE:
        Win32ErrorCodeDescription := 'The directory service failed to lock a tree in preparation for a tree deletion because the tree was in use.';
    Win32ErrorCodes.ERROR_DS_COULDNT_IDENTIFY_OBJECTS_FOR_TREE_DELETE:
        Win32ErrorCodeDescription := 'The directory service failed to identify the list of objects to delete while attempting a tree deletion.';
    Win32ErrorCodes.ERROR_DS_SAM_INIT_FAILURE:
        Win32ErrorCodeDescription := 'Security Accounts Manager initialization failed because of the following error: %1. Error Status: 0x%2. Click OK to shut down the system and reboot into Directory Services Restore Mode. Check the event log for detailed information.';
    Win32ErrorCodes.ERROR_DS_SENSITIVE_GROUP_VIOLATION:
        Win32ErrorCodeDescription :=
            'Only an administrator can modify the membership list of an administrative group.';
    Win32ErrorCodes.ERROR_DS_CANT_MOD_PRIMARYGROUPID:
        Win32ErrorCodeDescription :=
            'Cannot change the primary group ID of a domain controller account.';
    Win32ErrorCodes.ERROR_DS_ILLEGAL_BASE_SCHEMA_MOD:
        Win32ErrorCodeDescription := 'An attempt is made to modify the base schema.';
    Win32ErrorCodes.ERROR_DS_NONSAFE_SCHEMA_CHANGE:
        Win32ErrorCodeDescription := 'Adding a new mandatory attribute to an existing class, deleting one from an existing class, or adding an optional attribute to the special class Top that is not a backlink attribute (directly or through inheritance) is not allowed.';
    Win32ErrorCodes.ERROR_DS_SCHEMA_UPDATE_DISALLOWED:
        Win32ErrorCodeDescription :=
            'Schema update is not allowed on this DC because the DC is not the schema FSMO Role Owner.';
    Win32ErrorCodes.ERROR_DS_CANT_CREATE_UNDER_SCHEMA:
        Win32ErrorCodeDescription := 'An object of this class cannot be created under the schema container. You can only create attribute-schema and class-schema objects under the schema container.';
    Win32ErrorCodes.ERROR_DS_INSTALL_NO_SRC_SCH_VERSION:
        Win32ErrorCodeDescription := 'The replica/child install failed to get the objectVersion attribute on the schema container on the source DC. Either the attribute is missing on the schema container or the credentials supplied do not have permission to read it.';
    Win32ErrorCodes.ERROR_DS_INSTALL_NO_SCH_VERSION_IN_INIFILE:
        Win32ErrorCodeDescription := 'The replica/child install failed to read the objectVersion attribute in the SCHEMA section of the file schema.ini in the system32 directory.';
    Win32ErrorCodes.ERROR_DS_INVALID_GROUP_TYPE:
        Win32ErrorCodeDescription := 'The specified group type is invalid.';
    Win32ErrorCodes.ERROR_DS_NO_NEST_GLOBALGROUP_IN_MIXEDDOMAIN:
        Win32ErrorCodeDescription :=
            'Cannot nest global groups in a mixed domain if the group is security-enabled.';
    Win32ErrorCodes.ERROR_DS_NO_NEST_LOCALGROUP_IN_MIXEDDOMAIN:
        Win32ErrorCodeDescription :=
            'Cannot nest local groups in a mixed domain if the group is security-enabled.';
    Win32ErrorCodes.ERROR_DS_GLOBAL_CANT_HAVE_LOCAL_MEMBER:
        Win32ErrorCodeDescription := 'A global group cannot have a local group as a member.';
    Win32ErrorCodes.ERROR_DS_GLOBAL_CANT_HAVE_UNIVERSAL_MEMBER:
        Win32ErrorCodeDescription := 'A global group cannot have a universal group as a member.';
    Win32ErrorCodes.ERROR_DS_UNIVERSAL_CANT_HAVE_LOCAL_MEMBER:
        Win32ErrorCodeDescription := 'A universal group cannot have a local group as a member.';
    Win32ErrorCodes.ERROR_DS_GLOBAL_CANT_HAVE_CROSSDOMAIN_MEMBER:
        Win32ErrorCodeDescription := 'A global group cannot have a cross-domain member.';
    Win32ErrorCodes.ERROR_DS_LOCAL_CANT_HAVE_CROSSDOMAIN_LOCAL_MEMBER:
        Win32ErrorCodeDescription :=
            'A local group cannot have another cross-domain local group as a member.';
    Win32ErrorCodes.ERROR_DS_HAVE_PRIMARY_MEMBERS:
        Win32ErrorCodeDescription :=
            'A group with primary members cannot change to a security-disabled group.';
    Win32ErrorCodes.ERROR_DS_STRING_SD_CONVERSION_FAILED:
        Win32ErrorCodeDescription :=
            'The schema cache load failed to convert the string default SD on a class-schema object.';
    Win32ErrorCodes.ERROR_DS_NAMING_MASTER_GC:
        Win32ErrorCodeDescription := 'Only DSAs configured to be Global Catalog servers should be allowed to hold the Domain Naming Master FSMO role. (Applies only to Windows 2000 servers)';
    Win32ErrorCodes.ERROR_DS_LOOKUP_FAILURE:
        Win32ErrorCodeDescription :=
            'The DSA operation is unable to proceed because of a DNS lookup failure.';
    Win32ErrorCodes.ERROR_DS_COULDNT_UPDATE_SPNS:
        Win32ErrorCodeDescription := 'While processing a change to the DNS Host Name for an object, the Service Principal Name values could not be kept in sync.';
    Win32ErrorCodes.ERROR_DS_CANT_RETRIEVE_SD:
        Win32ErrorCodeDescription := 'The Security Descriptor attribute could not be read.';
    Win32ErrorCodes.ERROR_DS_KEY_NOT_UNIQUE:
        Win32ErrorCodeDescription :=
            'The object requested was not found, but an object with that key was found.';
    Win32ErrorCodes.ERROR_DS_WRONG_LINKED_ATT_SYNTAX:
        Win32ErrorCodeDescription := 'The syntax of the linked attributed being added is incorrect. Forward links can only have syntax 2.5.5.1, 2.5.5.7, and 2.5.5.14, and backlinks can only have syntax 2.5.5.1.';
    Win32ErrorCodes.ERROR_DS_SAM_NEED_BOOTKEY_PASSWORD:
        Win32ErrorCodeDescription := 'Security Account Manager needs to get the boot password.';
    Win32ErrorCodes.ERROR_DS_SAM_NEED_BOOTKEY_FLOPPY:
        Win32ErrorCodeDescription :=
            'Security Account Manager needs to get the boot key from floppy disk.';
    Win32ErrorCodes.ERROR_DS_CANT_START:
        Win32ErrorCodeDescription := 'Directory Service cannot start.';
    Win32ErrorCodes.ERROR_DS_INIT_FAILURE:
        Win32ErrorCodeDescription := 'Directory Services could not start.';
    Win32ErrorCodes.ERROR_DS_NO_PKT_PRIVACY_ON_CONNECTION:
        Win32ErrorCodeDescription :=
            'The connection between client and server requires packet privacy or better.';
    Win32ErrorCodes.ERROR_DS_SOURCE_DOMAIN_IN_FOREST:
        Win32ErrorCodeDescription :=
            'The source domain may not be in the same forest as destination.';
    Win32ErrorCodes.ERROR_DS_DESTINATION_DOMAIN_NOT_IN_FOREST:
        Win32ErrorCodeDescription := 'The destination domain must be in the forest.';
    Win32ErrorCodes.ERROR_DS_DESTINATION_AUDITING_NOT_ENABLED:
        Win32ErrorCodeDescription :=
            'The operation requires that destination domain auditing be enabled.';
    Win32ErrorCodes.ERROR_DS_CANT_FIND_DC_FOR_SRC_DOMAIN:
        Win32ErrorCodeDescription := 'The operation couldnt locate a DC for the source domain.';
    Win32ErrorCodes.ERROR_DS_SRC_OBJ_NOT_GROUP_OR_USER:
        Win32ErrorCodeDescription := 'The source object must be a group or user.';
    Win32ErrorCodes.ERROR_DS_SRC_SID_EXISTS_IN_FOREST:
        Win32ErrorCodeDescription :=
            'The source objects SID already exists in destination forest.';
    Win32ErrorCodes.ERROR_DS_SRC_AND_DST_OBJECT_CLASS_MISMATCH:
        Win32ErrorCodeDescription := 'The source and destination object must be of the same type.';
    Win32ErrorCodes.ERROR_SAM_INIT_FAILURE:
        Win32ErrorCodeDescription := 'Security Accounts Manager initialization failed because of the following error: %1. Error Status: 0x%2. Click OK to shut down the system and reboot into Safe Mode. Check the event log for detailed information.';
    Win32ErrorCodes.ERROR_DS_DRA_SCHEMA_INFO_SHIP:
        Win32ErrorCodeDescription :=
            'Schema information could not be included in the replication request.';
    Win32ErrorCodes.ERROR_DS_DRA_SCHEMA_CONFLICT:
        Win32ErrorCodeDescription :=
            'The replication operation could not be completed due to a schema incompatibility.';
    Win32ErrorCodes.ERROR_DS_DRA_EARLIER_SCHEMA_CONLICT:
        Win32ErrorCodeDescription := 'The replication operation could not be completed due to a previous schema incompatibility.';
    Win32ErrorCodes.ERROR_DS_DRA_OBJ_NC_MISMATCH:
        Win32ErrorCodeDescription := 'The replication update could not be applied because either the source or the destination has not yet received information regarding a recent cross-domain move operation.';
    Win32ErrorCodes.ERROR_DS_NC_STILL_HAS_DSAS:
        Win32ErrorCodeDescription := 'The requested domain could not be deleted because there exist domain controllers that still host this domain.';
    Win32ErrorCodes.ERROR_DS_GC_REQUIRED:
        Win32ErrorCodeDescription :=
            'The requested operation can be performed only on a global catalog server.';
    Win32ErrorCodes.ERROR_DS_LOCAL_MEMBER_OF_LOCAL_ONLY:
        Win32ErrorCodeDescription :=
            'A local group can only be a member of other local groups in the same domain.';
    Win32ErrorCodes.ERROR_DS_NO_FPO_IN_UNIVERSAL_GROUPS:
        Win32ErrorCodeDescription :=
            'Foreign security principals cannot be members of universal groups.';
    Win32ErrorCodes.ERROR_DS_CANT_ADD_TO_GC:
        Win32ErrorCodeDescription :=
            'The attribute is not allowed to be replicated to the GC because of security reasons.';
    Win32ErrorCodes.ERROR_DS_NO_CHECKPOINT_WITH_PDC:
        Win32ErrorCodeDescription := 'The checkpoint with the PDC could not be taken because there are too many modifications being processed currently.';
    Win32ErrorCodes.ERROR_DS_SOURCE_AUDITING_NOT_ENABLED:
        Win32ErrorCodeDescription :=
            'The operation requires that source domain auditing be enabled.';
    Win32ErrorCodes.ERROR_DS_CANT_CREATE_IN_NONDOMAIN_NC:
        Win32ErrorCodeDescription :=
            'Security principal objects can only be created inside domain naming contexts.';
    Win32ErrorCodes.ERROR_DS_INVALID_NAME_FOR_SPN:
        Win32ErrorCodeDescription := 'A Service Principal Name (SPN) could not be constructed because the provided hostname is not in the necessary format.';
    Win32ErrorCodes.ERROR_DS_FILTER_USES_CONTRUCTED_ATTRS:
        Win32ErrorCodeDescription := 'A Filter was passed that uses constructed attributes.';
    Win32ErrorCodes.ERROR_DS_UNICODEPWD_NOT_IN_QUOTES:
        Win32ErrorCodeDescription :=
            'The unicodePwd attribute value must be enclosed in double quotes.';
    Win32ErrorCodes.ERROR_DS_MACHINE_ACCOUNT_QUOTA_EXCEEDED:
        Win32ErrorCodeDescription := 'Your computer could not be joined to the domain. You have exceeded the maximum number of computer accounts you are allowed to create in this domain. Contact your system administrator to have this limit reset or increased.';
    Win32ErrorCodes.ERROR_DS_MUST_BE_RUN_ON_DST_DC:
        Win32ErrorCodeDescription :=
            'For security reasons, the operation must be run on the destination DC.';
    Win32ErrorCodes.ERROR_DS_SRC_DC_MUST_BE_SP4_OR_GREATER:
        Win32ErrorCodeDescription :=
            'For security reasons, the source DC must be NT4SP4 or greater.';
    Win32ErrorCodes.ERROR_DS_CANT_TREE_DELETE_CRITICAL_OBJ:
        Win32ErrorCodeDescription := 'Critical Directory Service System objects cannot be deleted during tree delete operations. The tree delete may have been partially performed.';
    Win32ErrorCodes.ERROR_DS_INIT_FAILURE_CONSOLE:
        Win32ErrorCodeDescription := 'Directory Services could not start because of the following error: %1. Error Status: 0x%2. Please click OK to shutdown the system. You can use the recovery console to diagnose the system further.';
    Win32ErrorCodes.ERROR_DS_SAM_INIT_FAILURE_CONSOLE:
        Win32ErrorCodeDescription := 'Security Accounts Manager initialization failed because of the following error: %1. Error Status: 0x%2. Please click OK to shutdown the system. You can use the recovery console to diagnose the system further.';
    Win32ErrorCodes.ERROR_DS_FOREST_VERSION_TOO_HIGH:
        Win32ErrorCodeDescription := 'This version of Windows is too old to support the current directory forest behavior. You must upgrade the operating system on this server before it can become a domain controller in this forest.';
    Win32ErrorCodes.ERROR_DS_DOMAIN_VERSION_TOO_HIGH:
        Win32ErrorCodeDescription := 'This version of Windows is too old to support the current domain behavior. You must upgrade the operating system on this server before it can become a domain controller in this domain.';
    Win32ErrorCodes.ERROR_DS_FOREST_VERSION_TOO_LOW:
        Win32ErrorCodeDescription := 'This version of Windows no longer supports the behavior version in use in this directory forest. You must advance the forest behavior version before this server can become a domain controller in the forest.';
    Win32ErrorCodes.ERROR_DS_DOMAIN_VERSION_TOO_LOW:
        Win32ErrorCodeDescription := 'This version of Windows no longer supports the behavior version in use in this domain. You must advance the domain behavior version before this server can become a domain controller in the domain.';
    Win32ErrorCodes.ERROR_DS_INCOMPATIBLE_VERSION:
        Win32ErrorCodeDescription :=
            'The version of Windows is incompatible with the behavior version of the domain or forest.';
    Win32ErrorCodes.ERROR_DS_LOW_DSA_VERSION:
        Win32ErrorCodeDescription := 'The behavior version cannot be increased to the requested value because Domain Controllers still exist with versions lower than the requested value.';
    Win32ErrorCodes.ERROR_DS_NO_BEHAVIOR_VERSION_IN_MIXEDDOMAIN:
        Win32ErrorCodeDescription := 'The behavior version value cannot be increased while the domain is still in mixed domain mode. You must first change the domain to native mode before increasing the behavior version.';
    Win32ErrorCodes.ERROR_DS_NOT_SUPPORTED_SORT_ORDER:
        Win32ErrorCodeDescription := 'The sort order requested is not supported.';
    Win32ErrorCodes.ERROR_DS_NAME_NOT_UNIQUE:
        Win32ErrorCodeDescription := 'Found an object with a non unique name.';
    Win32ErrorCodes.ERROR_DS_MACHINE_ACCOUNT_CREATED_PRENT4:
        Win32ErrorCodeDescription :=
            'The machine account was created pre-NT4. The account needs to be recreated.';
    Win32ErrorCodes.ERROR_DS_OUT_OF_VERSION_STORE:
        Win32ErrorCodeDescription := 'The database is out of version store.';
    Win32ErrorCodes.ERROR_DS_INCOMPATIBLE_CONTROLS_USED:
        Win32ErrorCodeDescription :=
            'Unable to continue operation because multiple conflicting controls were used.';
    Win32ErrorCodes.ERROR_DS_NO_REF_DOMAIN:
        Win32ErrorCodeDescription :=
            'Unable to find a valid security descriptor reference domain for this partition.';
    Win32ErrorCodes.ERROR_DS_RESERVED_LINK_ID:
        Win32ErrorCodeDescription := 'Schema update failed: The link identifier is reserved.';
    Win32ErrorCodes.ERROR_DS_LINK_ID_NOT_AVAILABLE:
        Win32ErrorCodeDescription :=
            'Schema update failed: There are no link identifiers available.';
    Win32ErrorCodes.ERROR_DS_AG_CANT_HAVE_UNIVERSAL_MEMBER:
        Win32ErrorCodeDescription :=
            'An account group can not have a universal group as a member.';
    Win32ErrorCodes.ERROR_DS_MODIFYDN_DISALLOWED_BY_INSTANCE_TYPE:
        Win32ErrorCodeDescription :=
            'Rename or move operations on naming context heads or read-only objects are not allowed.';
    Win32ErrorCodes.ERROR_DS_NO_OBJECT_MOVE_IN_SCHEMA_NC:
        Win32ErrorCodeDescription :=
            'Move operations on objects in the schema naming context are not allowed.';
    Win32ErrorCodes.ERROR_DS_MODIFYDN_DISALLOWED_BY_FLAG:
        Win32ErrorCodeDescription := 'A system flag has been set on the object and does not allow the object to be moved or renamed.';
    Win32ErrorCodes.ERROR_DS_MODIFYDN_WRONG_GRANDPARENT:
        Win32ErrorCodeDescription := 'This object is not allowed to change its grandparent container. Moves are not forbidden on this object, but are restricted to sibling containers.';
    Win32ErrorCodes.ERROR_DS_NAME_ERROR_TRUST_REFERRAL:
        Win32ErrorCodeDescription :=
            'Unable to resolve completely, a referral to another forest is generated.';
    Win32ErrorCodes.ERROR_NOT_SUPPORTED_ON_STANDARD_SERVER:
        Win32ErrorCodeDescription := 'The requested action is not supported on standard server.';
    Win32ErrorCodes.ERROR_DS_CANT_ACCESS_REMOTE_PART_OF_AD:
        Win32ErrorCodeDescription := 'Could not access a partition of the Active Directory located on a remote server. Make sure at least one server is running for the partition in question.';
    Win32ErrorCodes.ERROR_DS_CR_IMPOSSIBLE_TO_VALIDATE_V2:
        Win32ErrorCodeDescription := 'The directory cant validate the proposed naming context (or partition) name because it doesnt hold a replica nor can it contact a replica of the naming context above the proposed naming context.';
    Win32ErrorCodes.ERROR_DS_THREAD_LIMIT_EXCEEDED:
        Win32ErrorCodeDescription := 'The thread limit for this request was exceeded.';
    Win32ErrorCodes.ERROR_DS_NOT_CLOSEST:
        Win32ErrorCodeDescription := 'The Global catalog server is not in the closet site.';
    Win32ErrorCodes.DNS_ERROR_RCODE_FORMAT_ERROR:
        Win32ErrorCodeDescription := 'DNS server unable to interpret format.';
    Win32ErrorCodes.DNS_ERROR_RCODE_SERVER_FAILURE:
        Win32ErrorCodeDescription := 'DNS server failure.';
    Win32ErrorCodes.DNS_ERROR_RCODE_NAME_ERROR:
        Win32ErrorCodeDescription := 'DNS name does not exist.';
    Win32ErrorCodes.DNS_ERROR_RCODE_NOT_IMPLEMENTED:
        Win32ErrorCodeDescription := 'DNS request not supported by name server.';
    Win32ErrorCodes.DNS_ERROR_RCODE_REFUSED:
        Win32ErrorCodeDescription := 'DNS operation refused.';
    Win32ErrorCodes.DNS_ERROR_RCODE_YXDOMAIN:
        Win32ErrorCodeDescription := 'DNS name that ought not exist, does exist.';
    Win32ErrorCodes.DNS_ERROR_RCODE_YXRRSET:
        Win32ErrorCodeDescription := 'DNS RR set that ought not exist, does exist.';
    Win32ErrorCodes.DNS_ERROR_RCODE_NXRRSET:
        Win32ErrorCodeDescription := 'DNS RR set that ought to exist, does not exist.';
    Win32ErrorCodes.DNS_ERROR_RCODE_NOTAUTH:
        Win32ErrorCodeDescription := 'DNS server not authoritative for zone.';
    Win32ErrorCodes.DNS_ERROR_RCODE_NOTZONE:
        Win32ErrorCodeDescription := 'DNS name in update or prereq is not in zone.';
    Win32ErrorCodes.DNS_ERROR_RCODE_BADSIG:
        Win32ErrorCodeDescription := 'DNS signature failed to verify.';
    Win32ErrorCodes.DNS_ERROR_RCODE_BADKEY:
        Win32ErrorCodeDescription := 'DNS bad key.';
    Win32ErrorCodes.DNS_ERROR_RCODE_BADTIME:
        Win32ErrorCodeDescription := 'DNS signature validity expired.';
    Win32ErrorCodes.DNS_INFO_NO_RECORDS:
        Win32ErrorCodeDescription := 'No records found for given DNS query.';
    Win32ErrorCodes.DNS_ERROR_BAD_PACKET:
        Win32ErrorCodeDescription := 'Bad DNS packet.';
    Win32ErrorCodes.DNS_ERROR_NO_PACKET:
        Win32ErrorCodeDescription := 'No DNS packet.';
    Win32ErrorCodes.DNS_ERROR_RCODE:
        Win32ErrorCodeDescription := 'DNS error, check rcode.';
    Win32ErrorCodes.DNS_ERROR_UNSECURE_PACKET:
        Win32ErrorCodeDescription := 'Unsecured DNS packet.';
    Win32ErrorCodes.DNS_ERROR_INVALID_TYPE:
        Win32ErrorCodeDescription := 'Invalid DNS type.';
    Win32ErrorCodes.DNS_ERROR_INVALID_IP_ADDRESS:
        Win32ErrorCodeDescription := 'Invalid IP address.';
    Win32ErrorCodes.DNS_ERROR_INVALID_PROPERTY:
        Win32ErrorCodeDescription := 'Invalid property.';
    Win32ErrorCodes.DNS_ERROR_TRY_AGAIN_LATER:
        Win32ErrorCodeDescription := 'Try DNS operation again later.';
    Win32ErrorCodes.DNS_ERROR_NOT_UNIQUE:
        Win32ErrorCodeDescription := 'Record for given name and type is not unique.';
    Win32ErrorCodes.DNS_ERROR_NON_RFC_NAME:
        Win32ErrorCodeDescription := 'DNS name does not comply with RFC specifications.';
    Win32ErrorCodes.DNS_STATUS_FQDN:
        Win32ErrorCodeDescription := 'DNS name is a fully-qualified DNS name.';
    Win32ErrorCodes.DNS_STATUS_DOTTED_NAME:
        Win32ErrorCodeDescription := 'DNS name is dotted (multi-label).';
    Win32ErrorCodes.DNS_STATUS_SINGLE_PART_NAME:
        Win32ErrorCodeDescription := 'DNS name is a single-part name.';
    Win32ErrorCodes.DNS_ERROR_INVALID_NAME_CHAR:
        Win32ErrorCodeDescription := 'DSN name contains an invalid character.';
    Win32ErrorCodes.DNS_ERROR_NUMERIC_NAME:
        Win32ErrorCodeDescription := 'DNS name is entirely numeric.';
    Win32ErrorCodes.DNS_ERROR_ZONE_DOES_NOT_EXIST:
        Win32ErrorCodeDescription := 'DNS zone does not exist.';
    Win32ErrorCodes.DNS_ERROR_NO_ZONE_INFO:
        Win32ErrorCodeDescription := 'DNS zone information not available.';
    Win32ErrorCodes.DNS_ERROR_INVALID_ZONE_OPERATION:
        Win32ErrorCodeDescription := 'Invalid operation for DNS zone.';
    Win32ErrorCodes.DNS_ERROR_ZONE_CONFIGURATION_ERROR:
        Win32ErrorCodeDescription := 'Invalid DNS zone configuration.';
    Win32ErrorCodes.DNS_ERROR_ZONE_HAS_NO_SOA_RECORD:
        Win32ErrorCodeDescription := 'DNS zone has no start of authority (SOA) record.';
    Win32ErrorCodes.DNS_ERROR_ZONE_HAS_NO_NS_RECORDS:
        Win32ErrorCodeDescription := 'DNS zone has no name server (NS) record.';
    Win32ErrorCodes.DNS_ERROR_ZONE_LOCKED:
        Win32ErrorCodeDescription := 'DNS zone is locked.';
    Win32ErrorCodes.DNS_ERROR_ZONE_CREATION_FAILED:
        Win32ErrorCodeDescription := 'DNS zone creation failed.';
    Win32ErrorCodes.DNS_ERROR_ZONE_ALREADY_EXISTS:
        Win32ErrorCodeDescription := 'DNS zone already exists.';
    Win32ErrorCodes.DNS_ERROR_AUTOZONE_ALREADY_EXISTS:
        Win32ErrorCodeDescription := 'DNS automatic zone already exists.';
    Win32ErrorCodes.DNS_ERROR_INVALID_ZONE_TYPE:
        Win32ErrorCodeDescription := 'Invalid DNS zone type.';
    Win32ErrorCodes.DNS_ERROR_SECONDARY_REQUIRES_MASTER_IP:
        Win32ErrorCodeDescription := 'Secondary DNS zone requires master IP address.';
    Win32ErrorCodes.DNS_ERROR_ZONE_NOT_SECONDARY:
        Win32ErrorCodeDescription := 'DNS zone not secondary.';
    Win32ErrorCodes.DNS_ERROR_NEED_SECONDARY_ADDRESSES:
        Win32ErrorCodeDescription := 'Need secondary IP address.';
    Win32ErrorCodes.DNS_ERROR_WINS_INIT_FAILED:
        Win32ErrorCodeDescription := 'WINS initialization failed.';
    Win32ErrorCodes.DNS_ERROR_NEED_WINS_SERVERS:
        Win32ErrorCodeDescription := 'Need WINS servers.';
    Win32ErrorCodes.DNS_ERROR_NBSTAT_INIT_FAILED:
        Win32ErrorCodeDescription := 'NBTSTAT initialization call failed.';
    Win32ErrorCodes.DNS_ERROR_SOA_DELETE_INVALID:
        Win32ErrorCodeDescription := 'Invalid delete of start of authority (SOA)';
    Win32ErrorCodes.DNS_ERROR_FORWARDER_ALREADY_EXISTS:
        Win32ErrorCodeDescription := 'A conditional forwarding zone already exists for that name.';
    Win32ErrorCodes.DNS_ERROR_PRIMARY_REQUIRES_DATAFILE:
        Win32ErrorCodeDescription := 'Primary DNS zone requires datafile.';
    Win32ErrorCodes.DNS_ERROR_INVALID_DATAFILE_NAME:
        Win32ErrorCodeDescription := 'Invalid datafile name for DNS zone.';
    Win32ErrorCodes.DNS_ERROR_DATAFILE_OPEN_FAILURE:
        Win32ErrorCodeDescription := 'Failed to open datafile for DNS zone.';
    Win32ErrorCodes.DNS_ERROR_FILE_WRITEBACK_FAILED:
        Win32ErrorCodeDescription := 'Failed to write datafile for DNS zone.';
    Win32ErrorCodes.DNS_ERROR_DATAFILE_PARSING:
        Win32ErrorCodeDescription := 'Failure while reading datafile for DNS zone.';
    Win32ErrorCodes.DNS_ERROR_RECORD_DOES_NOT_EXIST:
        Win32ErrorCodeDescription := 'DNS record does not exist.';
    Win32ErrorCodes.DNS_ERROR_RECORD_FORMAT:
        Win32ErrorCodeDescription := 'DNS record format error.';
    Win32ErrorCodes.DNS_ERROR_NODE_CREATION_FAILED:
        Win32ErrorCodeDescription := 'Node creation failure in DNS.';
    Win32ErrorCodes.DNS_ERROR_UNKNOWN_RECORD_TYPE:
        Win32ErrorCodeDescription := 'Unknown DNS record type.';
    Win32ErrorCodes.DNS_ERROR_RECORD_TIMED_OUT:
        Win32ErrorCodeDescription := 'DNS record timed out.';
    Win32ErrorCodes.DNS_ERROR_NAME_NOT_IN_ZONE:
        Win32ErrorCodeDescription := 'Name not in DNS zone.';
    Win32ErrorCodes.DNS_ERROR_CNAME_LOOP:
        Win32ErrorCodeDescription := 'CNAME loop detected.';
    Win32ErrorCodes.DNS_ERROR_NODE_IS_CNAME:
        Win32ErrorCodeDescription := 'Node is a CNAME DNS record.';
    Win32ErrorCodes.DNS_ERROR_CNAME_COLLISION:
        Win32ErrorCodeDescription := 'A CNAME record already exists for given name.';
    Win32ErrorCodes.DNS_ERROR_RECORD_ONLY_AT_ZONE_ROOT:
        Win32ErrorCodeDescription := 'Record only at DNS zone root.';
    Win32ErrorCodes.DNS_ERROR_RECORD_ALREADY_EXISTS:
        Win32ErrorCodeDescription := 'DNS record already exists.';
    Win32ErrorCodes.DNS_ERROR_SECONDARY_DATA:
        Win32ErrorCodeDescription := 'Secondary DNS zone data error.';
    Win32ErrorCodes.DNS_ERROR_NO_CREATE_CACHE_DATA:
        Win32ErrorCodeDescription := 'Could not create DNS cache data.';
    Win32ErrorCodes.DNS_ERROR_NAME_DOES_NOT_EXIST:
        Win32ErrorCodeDescription := 'DNS name does not exist.';
    Win32ErrorCodes.DNS_WARNING_PTR_CREATE_FAILED:
        Win32ErrorCodeDescription := 'Could not create pointer (PTR) record.';
    Win32ErrorCodes.DNS_WARNING_DOMAIN_UNDELETED:
        Win32ErrorCodeDescription := 'DNS domain was undeleted.';
    Win32ErrorCodes.DNS_ERROR_DS_UNAVAILABLE:
        Win32ErrorCodeDescription := 'The directory service is unavailable.';
    Win32ErrorCodes.DNS_ERROR_DS_ZONE_ALREADY_EXISTS:
        Win32ErrorCodeDescription := 'DNS zone already exists in the directory service.';
    Win32ErrorCodes.DNS_ERROR_NO_BOOTFILE_IF_DS_ZONE:
        Win32ErrorCodeDescription := 'DNS server not creating or reading the boot file for the directory service integrated DNS zone.';
    Win32ErrorCodes.DNS_INFO_AXFR_COMPLETE:
        Win32ErrorCodeDescription := 'DNS AXFR (zone transfer) complete.';
    Win32ErrorCodes.DNS_ERROR_AXFR:
        Win32ErrorCodeDescription := 'DNS zone transfer failed.';
    Win32ErrorCodes.DNS_INFO_ADDED_LOCAL_WINS:
        Win32ErrorCodeDescription := 'Added local WINS server.';
    Win32ErrorCodes.DNS_STATUS_CONTINUE_NEEDED:
        Win32ErrorCodeDescription := 'Secure update call needs to continue update request.';
    Win32ErrorCodes.DNS_ERROR_NO_TCPIP:
        Win32ErrorCodeDescription := 'TCP/IP network protocol not installed.';
    Win32ErrorCodes.DNS_ERROR_NO_DNS_SERVERS:
        Win32ErrorCodeDescription := 'No DNS servers configured for local system.';
    Win32ErrorCodes.DNS_ERROR_DP_DOES_NOT_EXIST:
        Win32ErrorCodeDescription := 'The specified directory partition does not exist.';
    Win32ErrorCodes.DNS_ERROR_DP_ALREADY_EXISTS:
        Win32ErrorCodeDescription := 'The specified directory partition already exists.';
    Win32ErrorCodes.DNS_ERROR_DP_NOT_ENLISTED:
        Win32ErrorCodeDescription :=
            'The DS is not enlisted in the specified directory partition.';
    Win32ErrorCodes.DNS_ERROR_DP_ALREADY_ENLISTED:
        Win32ErrorCodeDescription :=
            'The DS is already enlisted in the specified directory partition.';
    Win32ErrorCodes.WSAEINTR:
        Win32ErrorCodeDescription :=
            'A blocking operation was interrupted by a call to WSACancelBlockingCall.';
    Win32ErrorCodes.WSAEBADF:
        Win32ErrorCodeDescription := 'The file handle supplied is not valid.';
    Win32ErrorCodes.WSAEACCES:
        Win32ErrorCodeDescription :=
            'An attempt was made to access a socket in a way forbidden by its access permissions.';
    Win32ErrorCodes.WSAEFAULT:
        Win32ErrorCodeDescription := 'The system detected an invalid pointer address in attempting to use a pointer argument in a call.';
    Win32ErrorCodes.WSAEINVAL:
        Win32ErrorCodeDescription := 'An invalid argument was supplied.';
    Win32ErrorCodes.WSAEMFILE:
        Win32ErrorCodeDescription := 'Too many open sockets.';
    Win32ErrorCodes.WSAEWOULDBLOCK:
        Win32ErrorCodeDescription :=
            'A non-blocking socket operation could not be completed immediately.';
    Win32ErrorCodes.WSAEINPROGRESS:
        Win32ErrorCodeDescription := 'A blocking operation is currently executing.';
    Win32ErrorCodes.WSAEALREADY:
        Win32ErrorCodeDescription := 'An operation was attempted on a non-blocking socket that already had an operation in progress.';
    Win32ErrorCodes.WSAENOTSOCK:
        Win32ErrorCodeDescription :=
            'An operation was attempted on something that is not a socket.';
    Win32ErrorCodes.WSAEDESTADDRREQ:
        Win32ErrorCodeDescription :=
            'A required address was omitted from an operation on a socket.';
    Win32ErrorCodes.WSAEMSGSIZE:
        Win32ErrorCodeDescription := 'A message sent on a datagram socket was larger than the internal message buffer or some other network limit, or the buffer used to receive a datagram into was smaller than the datagram itself.';
    Win32ErrorCodes.WSAEPROTOTYPE:
        Win32ErrorCodeDescription := 'A protocol was specified in the socket function call that does not support the semantics of the socket type requested.';
    Win32ErrorCodes.WSAENOPROTOOPT:
        Win32ErrorCodeDescription := 'An unknown, invalid, or unsupported option or level was specified in a getsockopt or setsockopt call.';
    Win32ErrorCodes.WSAEPROTONOSUPPORT:
        Win32ErrorCodeDescription := 'The requested protocol has not been configured into the system, or no implementation for it exists.';
    Win32ErrorCodes.WSAESOCKTNOSUPPORT:
        Win32ErrorCodeDescription :=
            'The support for the specified socket type does not exist in this address family.';
    Win32ErrorCodes.WSAEOPNOTSUPP:
        Win32ErrorCodeDescription :=
            'The attempted operation is not supported for the type of object referenced.';
    Win32ErrorCodes.WSAEPFNOSUPPORT:
        Win32ErrorCodeDescription := 'The protocol family has not been configured into the system or no implementation for it exists.';
    Win32ErrorCodes.WSAEAFNOSUPPORT:
        Win32ErrorCodeDescription :=
            'An address incompatible with the requested protocol was used.';
    Win32ErrorCodes.WSAEADDRINUSE:
        Win32ErrorCodeDescription := 'Only one usage of each socket address (protocol/network address/port) is normally permitted.';
    Win32ErrorCodes.WSAEADDRNOTAVAIL:
        Win32ErrorCodeDescription := 'The requested address is not valid in its context.';
    Win32ErrorCodes.WSAENETDOWN:
        Win32ErrorCodeDescription := 'A socket operation encountered a dead network.';
    Win32ErrorCodes.WSAENETUNREACH:
        Win32ErrorCodeDescription := 'A socket operation was attempted to an unreachable network.';
    Win32ErrorCodes.WSAENETRESET:
        Win32ErrorCodeDescription := 'The connection has been broken due to keep-alive activity detecting a failure while the operation was in progress.';
    Win32ErrorCodes.WSAECONNABORTED:
        Win32ErrorCodeDescription :=
            'An established connection was aborted by the software in your host machine.';
    Win32ErrorCodes.WSAECONNRESET:
        Win32ErrorCodeDescription :=
            'An existing connection was forcibly closed by the remote host.';
    Win32ErrorCodes.WSAENOBUFS:
        Win32ErrorCodeDescription := 'An operation on a socket could not be performed because the system lacked sufficient buffer space or because a queue was full.';
    Win32ErrorCodes.WSAEISCONN:
        Win32ErrorCodeDescription := 'A connect request was made on an already connected socket.';
    Win32ErrorCodes.WSAENOTCONN:
        Win32ErrorCodeDescription := 'A request to send or receive data was disallowed because the socket is not connected and (when sending on a datagram socket using a sendto call) no address was supplied.';
    Win32ErrorCodes.WSAESHUTDOWN:
        Win32ErrorCodeDescription := 'A request to send or receive data was disallowed because the socket had already been shut down in that direction with a previous shutdown call.';
    Win32ErrorCodes.WSAETOOMANYREFS:
        Win32ErrorCodeDescription := 'Too many references to some kernel object.';
    Win32ErrorCodes.WSAETIMEDOUT:
        Win32ErrorCodeDescription := 'A connection attempt failed because the connected party did not properly respond after a period of time, or established connection failed because connected host has failed to respond.';
    Win32ErrorCodes.WSAECONNREFUSED:
        Win32ErrorCodeDescription :=
            'No connection could be made because the target machine actively refused it.';
    Win32ErrorCodes.WSAELOOP:
        Win32ErrorCodeDescription := 'Cannot translate name.';
    Win32ErrorCodes.WSAENAMETOOLONG:
        Win32ErrorCodeDescription := 'Name component or name was too long.';
    Win32ErrorCodes.WSAEHOSTDOWN:
        Win32ErrorCodeDescription :=
            'A socket operation failed because the destination host was down.';
    Win32ErrorCodes.WSAEHOSTUNREACH:
        Win32ErrorCodeDescription := 'A socket operation was attempted to an unreachable host.';
    Win32ErrorCodes.WSAENOTEMPTY:
        Win32ErrorCodeDescription := 'Cannot remove a directory that is not empty.';
    Win32ErrorCodes.WSAEPROCLIM:
        Win32ErrorCodeDescription := 'A Windows Sockets implementation may have a limit on the number of applications that may use it simultaneously.';
    Win32ErrorCodes.WSAEUSERS:
        Win32ErrorCodeDescription := 'Ran out of quota.';
    Win32ErrorCodes.WSAEDQUOT:
        Win32ErrorCodeDescription := 'Ran out of disk quota.';
    Win32ErrorCodes.WSAESTALE:
        Win32ErrorCodeDescription := 'File handle reference is no longer available.';
    Win32ErrorCodes.WSAEREMOTE:
        Win32ErrorCodeDescription := 'Item is not available locally.';
    Win32ErrorCodes.WSASYSNOTREADY:
        Win32ErrorCodeDescription := 'WSAStartup cannot function at this time because the underlying system it uses to provide network services is currently unavailable.';
    Win32ErrorCodes.WSAVERNOTSUPPORTED:
        Win32ErrorCodeDescription := 'The Windows Sockets version requested is not supported.';
    Win32ErrorCodes.WSANOTINITIALISED:
        Win32ErrorCodeDescription :=
            'Either the application has not called WSAStartup, or WSAStartup failed.';
    Win32ErrorCodes.WSAEDISCON:
        Win32ErrorCodeDescription := 'Returned by WSARecv or WSARecvFrom to indicate the remote party has initiated a graceful shutdown sequence.';
    Win32ErrorCodes.WSAENOMORE:
        Win32ErrorCodeDescription := 'No more results can be returned by WSALookupServiceNext.';
    Win32ErrorCodes.WSAECANCELLED:
        Win32ErrorCodeDescription := 'A call to WSALookupServiceEnd was made while this call was still processing. The call has been canceled.';
    Win32ErrorCodes.WSAEINVALIDPROCTABLE:
        Win32ErrorCodeDescription := 'The procedure call table is invalid.';
    Win32ErrorCodes.WSAEINVALIDPROVIDER:
        Win32ErrorCodeDescription := 'The requested service provider is invalid.';
    Win32ErrorCodes.WSAEPROVIDERFAILEDINIT:
        Win32ErrorCodeDescription :=
            'The requested service provider could not be loaded or initialized.';
    Win32ErrorCodes.WSASYSCALLFAILURE:
        Win32ErrorCodeDescription := 'A system call that should never fail has failed.';
    Win32ErrorCodes.WSASERVICE_NOT_FOUND:
        Win32ErrorCodeDescription :=
            'No such service is known. The service cannot be found in the specified name space.';
    Win32ErrorCodes.WSATYPE_NOT_FOUND:
        Win32ErrorCodeDescription := 'The specified class was not found.';
    Win32ErrorCodes.WSA_E_NO_MORE:
        Win32ErrorCodeDescription := 'No more results can be returned by WSALookupServiceNext.';
    Win32ErrorCodes.WSA_E_CANCELLED:
        Win32ErrorCodeDescription := 'A call to WSALookupServiceEnd was made while this call was still processing. The call has been canceled.';
    Win32ErrorCodes.WSAEREFUSED:
        Win32ErrorCodeDescription := 'A database query failed because it was actively refused.';
    Win32ErrorCodes.WSAHOST_NOT_FOUND:
        Win32ErrorCodeDescription := 'No such host is known.';
    Win32ErrorCodes.WSATRY_AGAIN:
        Win32ErrorCodeDescription := 'This is usually a temporary error during hostname resolution and means that the local server did not receive a response from an authoritative server.';
    Win32ErrorCodes.WSANO_RECOVERY:
        Win32ErrorCodeDescription := 'A non-recoverable error occurred during a database lookup.';
    Win32ErrorCodes.WSANO_DATA:
        Win32ErrorCodeDescription := 'The requested name is valid and was found in the database, but it does not have the correct associated data being resolved for.';
    Win32ErrorCodes.WSA_QOS_RECEIVERS:
        Win32ErrorCodeDescription := 'At least one reserve has arrived.';
    Win32ErrorCodes.WSA_QOS_SENDERS:
        Win32ErrorCodeDescription := 'At least one path has arrived.';
    Win32ErrorCodes.WSA_QOS_NO_SENDERS:
        Win32ErrorCodeDescription := 'There are no senders.';
    Win32ErrorCodes.WSA_QOS_NO_RECEIVERS:
        Win32ErrorCodeDescription := 'There are no receivers.';
    Win32ErrorCodes.WSA_QOS_REQUEST_CONFIRMED:
        Win32ErrorCodeDescription := 'Reserve has been confirmed.';
    Win32ErrorCodes.WSA_QOS_ADMISSION_FAILURE:
        Win32ErrorCodeDescription := 'Error due to lack of resources.';
    Win32ErrorCodes.WSA_QOS_POLICY_FAILURE:
        Win32ErrorCodeDescription := 'Rejected for administrative reasons - bad credentials.';
    Win32ErrorCodes.WSA_QOS_BAD_STYLE:
        Win32ErrorCodeDescription := 'Unknown or conflicting style.';
    Win32ErrorCodes.WSA_QOS_BAD_OBJECT:
        Win32ErrorCodeDescription :=
            'Problem with some part of the filterspec or providerspecific buffer in general.';
    Win32ErrorCodes.WSA_QOS_TRAFFIC_CTRL_ERROR:
        Win32ErrorCodeDescription := 'Problem with some part of the flowspec.';
    Win32ErrorCodes.WSA_QOS_GENERIC_ERROR:
        Win32ErrorCodeDescription := 'General QOS error.';
    Win32ErrorCodes.WSA_QOS_ESERVICETYPE:
        Win32ErrorCodeDescription :=
            'An invalid or unrecognized service type was found in the flowspec.';
    Win32ErrorCodes.WSA_QOS_EFLOWSPEC:
        Win32ErrorCodeDescription :=
            'An invalid or inconsistent flowspec was found in the QOS structure.';
    Win32ErrorCodes.WSA_QOS_EPROVSPECBUF:
        Win32ErrorCodeDescription := 'Invalid QOS provider-specific buffer.';
    Win32ErrorCodes.WSA_QOS_EFILTERSTYLE:
        Win32ErrorCodeDescription := 'An invalid QOS filter style was used.';
    Win32ErrorCodes.WSA_QOS_EFILTERTYPE:
        Win32ErrorCodeDescription := 'An invalid QOS filter type was used.';
    Win32ErrorCodes.WSA_QOS_EFILTERCOUNT:
        Win32ErrorCodeDescription :=
            'An incorrect number of QOS FILTERSPECs were specified in the FLOWDESCRIPTOR.';
    Win32ErrorCodes.WSA_QOS_EOBJLENGTH:
        Win32ErrorCodeDescription := 'An object with an invalid ObjectLength field was specified in the QOS provider-specific buffer.';
    Win32ErrorCodes.WSA_QOS_EFLOWCOUNT:
        Win32ErrorCodeDescription :=
            'An incorrect number of flow descriptors was specified in the QOS structure.';
    Win32ErrorCodes.WSA_QOS_EUNKNOWNPSOBJ:
        Win32ErrorCodeDescription :=
            'An unrecognized object was found in the QOS provider-specific buffer.';
    Win32ErrorCodes.WSA_QOS_EPOLICYOBJ:
        Win32ErrorCodeDescription :=
            'An invalid policy object was found in the QOS provider-specific buffer.';
    Win32ErrorCodes.WSA_QOS_EFLOWDESC:
        Win32ErrorCodeDescription :=
            'An invalid QOS flow descriptor was found in the flow descriptor list.';
    Win32ErrorCodes.WSA_QOS_EPSFLOWSPEC:
        Win32ErrorCodeDescription :=
            'An invalid or inconsistent flowspec was found in the QOS provider-specific buffer.';
    Win32ErrorCodes.WSA_QOS_EPSFILTERSPEC:
        Win32ErrorCodeDescription :=
            'An invalid FILTERSPEC was found in the QOS provider-specific buffer.';
    Win32ErrorCodes.WSA_QOS_ESDMODEOBJ:
        Win32ErrorCodeDescription :=
            'An invalid shape discard mode object was found in the QOS provider-specific buffer.';
    Win32ErrorCodes.WSA_QOS_ESHAPERATEOBJ:
        Win32ErrorCodeDescription :=
            'An invalid shaping rate object was found in the QOS provider-specific buffer.';
    Win32ErrorCodes.WSA_QOS_RESERVED_PETYPE:
        Win32ErrorCodeDescription :=
            'A reserved policy element was found in the QOS provider-specific buffer.';
    Win32ErrorCodes.ERROR_SXS_SECTION_NOT_FOUND:
        Win32ErrorCodeDescription :=
            'The requested section was not present in the activation context.';
    Win32ErrorCodes.ERROR_SXS_CANT_GEN_ACTCTX:
        Win32ErrorCodeDescription := 'This application has failed to start because the application configuration is incorrect. Reinstalling the application may fix this problem.';
    Win32ErrorCodes.ERROR_SXS_INVALID_ACTCTXDATA_FORMAT:
        Win32ErrorCodeDescription := 'The application binding data format is invalid.';
    Win32ErrorCodes.ERROR_SXS_ASSEMBLY_NOT_FOUND:
        Win32ErrorCodeDescription := 'The referenced assembly is not installed on your system.';
    Win32ErrorCodes.ERROR_SXS_MANIFEST_FORMAT_ERROR:
        Win32ErrorCodeDescription :=
            'The manifest file does not begin with the required tag and format information.';
    Win32ErrorCodes.ERROR_SXS_MANIFEST_PARSE_ERROR:
        Win32ErrorCodeDescription := 'The manifest file contains one or more syntax errors.';
    Win32ErrorCodes.ERROR_SXS_ACTIVATION_CONTEXT_DISABLED:
        Win32ErrorCodeDescription :=
            'The application attempted to activate a disabled activation context.';
    Win32ErrorCodes.ERROR_SXS_KEY_NOT_FOUND:
        Win32ErrorCodeDescription :=
            'The requested lookup key was not found in any active activation context.';
    Win32ErrorCodes.ERROR_SXS_VERSION_CONFLICT:
        Win32ErrorCodeDescription := 'A component version required by the application conflicts with another component version already active.';
    Win32ErrorCodes.ERROR_SXS_WRONG_SECTION_TYPE:
        Win32ErrorCodeDescription :=
            'The type requested activation context section does not match the query API used.';
    Win32ErrorCodes.ERROR_SXS_THREAD_QUERIES_DISABLED:
        Win32ErrorCodeDescription := 'Lack of system resources has required isolated activation to be disabled for the current thread of execution.';
    Win32ErrorCodes.ERROR_SXS_PROCESS_DEFAULT_ALREADY_SET:
        Win32ErrorCodeDescription := 'An attempt to set the process default activation context failed because the process default activation context was already set.';
    Win32ErrorCodes.ERROR_SXS_UNKNOWN_ENCODING_GROUP:
        Win32ErrorCodeDescription := 'The encoding group identifier specified is not recognized.';
    Win32ErrorCodes.ERROR_SXS_UNKNOWN_ENCODING:
        Win32ErrorCodeDescription := 'The encoding requested is not recognized.';
    Win32ErrorCodes.ERROR_SXS_INVALID_XML_NAMESPACE_URI:
        Win32ErrorCodeDescription := 'The manifest contains a reference to an invalid URI.';
    Win32ErrorCodes.ERROR_SXS_ROOT_MANIFEST_DEPENDENCY_NOT_INSTALLED:
        Win32ErrorCodeDescription := 'The application manifest contains a reference to a dependent assembly which is not installed.';
    Win32ErrorCodes.ERROR_SXS_LEAF_MANIFEST_DEPENDENCY_NOT_INSTALLED:
        Win32ErrorCodeDescription := 'The manifest for an assembly used by the application has a reference to a dependent assembly which is not installed.';
    Win32ErrorCodes.ERROR_SXS_INVALID_ASSEMBLY_IDENTITY_ATTRIBUTE:
        Win32ErrorCodeDescription :=
            'The manifest contains an attribute for the assembly identity which is not valid.';
    Win32ErrorCodes.ERROR_SXS_MANIFEST_MISSING_REQUIRED_DEFAULT_NAMESPACE:
        Win32ErrorCodeDescription := 'The manifest is missing the required default namespace specification on the assembly element.';
    Win32ErrorCodes.ERROR_SXS_MANIFEST_INVALID_REQUIRED_DEFAULT_NAMESPACE:
        Win32ErrorCodeDescription := 'The manifest has a default namespace specified on the assembly element but its value is not "urn:schemas-microsoft-com:asm.v1".';
    Win32ErrorCodes.ERROR_SXS_PRIVATE_MANIFEST_CROSS_PATH_WITH_REPARSE_POINT:
        Win32ErrorCodeDescription :=
            'The private manifest probe has crossed the reparse-point-associated path.';
    Win32ErrorCodes.ERROR_SXS_DUPLICATE_DLL_NAME:
        Win32ErrorCodeDescription := 'Two or more components referenced directly or indirectly by the application manifest have files by the same name.';
    Win32ErrorCodes.ERROR_SXS_DUPLICATE_WINDOWCLASS_NAME:
        Win32ErrorCodeDescription := 'Two or more components referenced directly or indirectly by the application manifest have window classes with the same name.';
    Win32ErrorCodes.ERROR_SXS_DUPLICATE_CLSID:
        Win32ErrorCodeDescription := 'Two or more components referenced directly or indirectly by the application manifest have the same COM server CLSIDs.';
    Win32ErrorCodes.ERROR_SXS_DUPLICATE_IID:
        Win32ErrorCodeDescription := 'Two or more components referenced directly or indirectly by the application manifest have proxies for the same COM interface IIDs.';
    Win32ErrorCodes.ERROR_SXS_DUPLICATE_TLBID:
        Win32ErrorCodeDescription := 'Two or more components referenced directly or indirectly by the application manifest have the same COM type library TLBIDs.';
    Win32ErrorCodes.ERROR_SXS_DUPLICATE_PROGID:
        Win32ErrorCodeDescription := 'Two or more components referenced directly or indirectly by the application manifest have the same COM ProgIDs.';
    Win32ErrorCodes.ERROR_SXS_DUPLICATE_ASSEMBLY_NAME:
        Win32ErrorCodeDescription := 'Two or more components referenced directly or indirectly by the application manifest are different versions of the same component which is not permitted.';
    Win32ErrorCodes.ERROR_SXS_FILE_HASH_MISMATCH:
        Win32ErrorCodeDescription := 'A components file does not match the verification information present in the component manifest.';
    Win32ErrorCodes.ERROR_SXS_POLICY_PARSE_ERROR:
        Win32ErrorCodeDescription := 'The policy manifest contains one or more syntax errors.';
    Win32ErrorCodes.ERROR_SXS_XML_E_MISSINGQUOTE:
        Win32ErrorCodeDescription := 'Manifest Parse Error : A string literal was expected, but no opening quote character was found.';
    Win32ErrorCodes.ERROR_SXS_XML_E_COMMENTSYNTAX:
        Win32ErrorCodeDescription :=
            'Manifest Parse Error : Incorrect syntax was used in a comment.';
    Win32ErrorCodes.ERROR_SXS_XML_E_BADSTARTNAMECHAR:
        Win32ErrorCodeDescription :=
            'Manifest Parse Error : A name was started with an invalid character.';
    Win32ErrorCodes.ERROR_SXS_XML_E_BADNAMECHAR:
        Win32ErrorCodeDescription :=
            'Manifest Parse Error : A name contained an invalid character.';
    Win32ErrorCodes.ERROR_SXS_XML_E_BADCHARINSTRING:
        Win32ErrorCodeDescription :=
            'Manifest Parse Error : A string literal contained an invalid character.';
    Win32ErrorCodes.ERROR_SXS_XML_E_XMLDECLSYNTAX:
        Win32ErrorCodeDescription :=
            'Manifest Parse Error : Invalid syntax for an XML declaration.';
    Win32ErrorCodes.ERROR_SXS_XML_E_BADCHARDATA:
        Win32ErrorCodeDescription :=
            'Manifest Parse Error : An invalid character was found in text content.';
    Win32ErrorCodes.ERROR_SXS_XML_E_MISSINGWHITESPACE:
        Win32ErrorCodeDescription := 'Manifest Parse Error : Required white space was missing.';
    Win32ErrorCodes.ERROR_SXS_XML_E_EXPECTINGTAGEND:
        Win32ErrorCodeDescription := 'Manifest Parse Error : The character &gt; was expected.';
    Win32ErrorCodes.ERROR_SXS_XML_E_MISSINGSEMICOLON:
        Win32ErrorCodeDescription := 'Manifest Parse Error : A semi colon character was expected.';
    Win32ErrorCodes.ERROR_SXS_XML_E_UNBALANCEDPAREN:
        Win32ErrorCodeDescription := 'Manifest Parse Error : Unbalanced parentheses.';
    Win32ErrorCodes.ERROR_SXS_XML_E_INTERNALERROR:
        Win32ErrorCodeDescription := 'Manifest Parse Error : Internal error.';
    Win32ErrorCodes.ERROR_SXS_XML_E_UNEXPECTED_WHITESPACE:
        Win32ErrorCodeDescription :=
            'Manifest Parse Error : White space is not allowed at this location.';
    Win32ErrorCodes.ERROR_SXS_XML_E_INCOMPLETE_ENCODING:
        Win32ErrorCodeDescription :=
            'Manifest Parse Error : End of file reached in invalid state for current encoding.';
    Win32ErrorCodes.ERROR_SXS_XML_E_MISSING_PAREN:
        Win32ErrorCodeDescription := 'Manifest Parse Error : Missing parenthesis.';
    Win32ErrorCodes.ERROR_SXS_XML_E_EXPECTINGCLOSEQUOTE:
        Win32ErrorCodeDescription :=
            'Manifest Parse Error : A single or double closing quote character (\ or \") is missing.';
    Win32ErrorCodes.ERROR_SXS_XML_E_MULTIPLE_COLONS:
        Win32ErrorCodeDescription :=
            'Manifest Parse Error : Multiple colons are not allowed in a name.';
    Win32ErrorCodes.ERROR_SXS_XML_E_INVALID_DECIMAL:
        Win32ErrorCodeDescription := 'Manifest Parse Error : Invalid character for decimal digit.';
    Win32ErrorCodes.ERROR_SXS_XML_E_INVALID_HEXIDECIMAL:
        Win32ErrorCodeDescription :=
            'Manifest Parse Error : Invalid character for hexadecimal digit.';
    Win32ErrorCodes.ERROR_SXS_XML_E_INVALID_UNICODE:
        Win32ErrorCodeDescription :=
            'Manifest Parse Error : Invalid Unicode character value for this platform.';
    Win32ErrorCodes.ERROR_SXS_XML_E_WHITESPACEORQUESTIONMARK:
        Win32ErrorCodeDescription := 'Manifest Parse Error : Expecting white space or ?.';
    Win32ErrorCodes.ERROR_SXS_XML_E_UNEXPECTEDENDTAG:
        Win32ErrorCodeDescription :=
            'Manifest Parse Error : End tag was not expected at this location.';
    Win32ErrorCodes.ERROR_SXS_XML_E_UNCLOSEDTAG:
        Win32ErrorCodeDescription :=
            'Manifest Parse Error : The following tags were not closed: %1.';
    Win32ErrorCodes.ERROR_SXS_XML_E_DUPLICATEATTRIBUTE:
        Win32ErrorCodeDescription := 'Manifest Parse Error : Duplicate attribute.';
    Win32ErrorCodes.ERROR_SXS_XML_E_MULTIPLEROOTS:
        Win32ErrorCodeDescription :=
            'Manifest Parse Error : Only one top level element is allowed in an XML document.';
    Win32ErrorCodes.ERROR_SXS_XML_E_INVALIDATROOTLEVEL:
        Win32ErrorCodeDescription :=
            'Manifest Parse Error : Invalid at the top level of the document.';
    Win32ErrorCodes.ERROR_SXS_XML_E_BADXMLDECL:
        Win32ErrorCodeDescription := 'Manifest Parse Error : Invalid XML declaration.';
    Win32ErrorCodes.ERROR_SXS_XML_E_MISSINGROOT:
        Win32ErrorCodeDescription :=
            'Manifest Parse Error : XML document must have a top level element.';
    Win32ErrorCodes.ERROR_SXS_XML_E_UNEXPECTEDEOF:
        Win32ErrorCodeDescription := 'Manifest Parse Error : Unexpected end of file.';
    Win32ErrorCodes.ERROR_SXS_XML_E_BADPEREFINSUBSET:
        Win32ErrorCodeDescription := 'Manifest Parse Error : Parameter entities cannot be used inside markup declarations in an internal subset.';
    Win32ErrorCodes.ERROR_SXS_XML_E_UNCLOSEDSTARTTAG:
        Win32ErrorCodeDescription := 'Manifest Parse Error : Element was not closed.';
    Win32ErrorCodes.ERROR_SXS_XML_E_UNCLOSEDENDTAG:
        Win32ErrorCodeDescription :=
            'Manifest Parse Error : End element was missing the character &gt;.';
    Win32ErrorCodes.ERROR_SXS_XML_E_UNCLOSEDSTRING:
        Win32ErrorCodeDescription := 'Manifest Parse Error : A string literal was not closed.';
    Win32ErrorCodes.ERROR_SXS_XML_E_UNCLOSEDCOMMENT:
        Win32ErrorCodeDescription := 'Manifest Parse Error : A comment was not closed.';
    Win32ErrorCodes.ERROR_SXS_XML_E_UNCLOSEDDECL:
        Win32ErrorCodeDescription := 'Manifest Parse Error : A declaration was not closed.';
    Win32ErrorCodes.ERROR_SXS_XML_E_UNCLOSEDCDATA:
        Win32ErrorCodeDescription := 'Manifest Parse Error : A CDATA section was not closed.';
    Win32ErrorCodes.ERROR_SXS_XML_E_RESERVEDNAMESPACE:
        Win32ErrorCodeDescription := 'Manifest Parse Error : The namespace prefix is not allowed to start with the reserved string "xml".';
    Win32ErrorCodes.ERROR_SXS_XML_E_INVALIDENCODING:
        Win32ErrorCodeDescription :=
            'Manifest Parse Error : System does not support the specified encoding.';
    Win32ErrorCodes.ERROR_SXS_XML_E_INVALIDSWITCH:
        Win32ErrorCodeDescription :=
            'Manifest Parse Error : Switch from current encoding to specified encoding not supported.';
    Win32ErrorCodes.ERROR_SXS_XML_E_BADXMLCASE:
        Win32ErrorCodeDescription :=
            'Manifest Parse Error : The name xml is reserved and must be lower case.';
    Win32ErrorCodes.ERROR_SXS_XML_E_INVALID_STANDALONE:
        Win32ErrorCodeDescription :=
            'Manifest Parse Error : The standalone attribute must have the value yes or no.';
    Win32ErrorCodes.ERROR_SXS_XML_E_UNEXPECTED_STANDALONE:
        Win32ErrorCodeDescription :=
            'Manifest Parse Error : The standalone attribute cannot be used in external entities.';
    Win32ErrorCodes.ERROR_SXS_XML_E_INVALID_VERSION:
        Win32ErrorCodeDescription := 'Manifest Parse Error : Invalid version number.';
    Win32ErrorCodes.ERROR_SXS_XML_E_MISSINGEQUALS:
        Win32ErrorCodeDescription :=
            'Manifest Parse Error : Missing equals sign between attribute and attribute value.';
    Win32ErrorCodes.ERROR_IPSEC_QM_POLICY_EXISTS:
        Win32ErrorCodeDescription := 'The specified quick mode policy already exists.';
    Win32ErrorCodes.ERROR_IPSEC_QM_POLICY_NOT_FOUND:
        Win32ErrorCodeDescription := 'The specified quick mode policy was not found.';
    Win32ErrorCodes.ERROR_IPSEC_QM_POLICY_IN_USE:
        Win32ErrorCodeDescription := 'The specified quick mode policy is being used.';
    Win32ErrorCodes.ERROR_IPSEC_MM_POLICY_EXISTS:
        Win32ErrorCodeDescription := 'The specified main mode policy already exists.';
    Win32ErrorCodes.ERROR_IPSEC_MM_POLICY_NOT_FOUND:
        Win32ErrorCodeDescription := 'The specified main mode policy was not found.';
    Win32ErrorCodes.ERROR_IPSEC_MM_POLICY_IN_USE:
        Win32ErrorCodeDescription := 'The specified main mode policy is being used.';
    Win32ErrorCodes.ERROR_IPSEC_MM_FILTER_EXISTS:
        Win32ErrorCodeDescription := 'The specified main mode filter already exists.';
    Win32ErrorCodes.ERROR_IPSEC_MM_FILTER_NOT_FOUND:
        Win32ErrorCodeDescription := 'The specified main mode filter was not found.';
    Win32ErrorCodes.ERROR_IPSEC_TRANSPORT_FILTER_EXISTS:
        Win32ErrorCodeDescription := 'The specified transport mode filter already exists.';
    Win32ErrorCodes.ERROR_IPSEC_TRANSPORT_FILTER_NOT_FOUND:
        Win32ErrorCodeDescription := 'The specified transport mode filter does not exist.';
    Win32ErrorCodes.ERROR_IPSEC_MM_AUTH_EXISTS:
        Win32ErrorCodeDescription := 'The specified main mode authentication list exists.';
    Win32ErrorCodes.ERROR_IPSEC_MM_AUTH_NOT_FOUND:
        Win32ErrorCodeDescription := 'The specified main mode authentication list was not found.';
    Win32ErrorCodes.ERROR_IPSEC_MM_AUTH_IN_USE:
        Win32ErrorCodeDescription := 'The specified quick mode policy is being used.';
    Win32ErrorCodes.ERROR_IPSEC_DEFAULT_MM_POLICY_NOT_FOUND:
        Win32ErrorCodeDescription := 'The specified main mode policy was not found.';
    Win32ErrorCodes.ERROR_IPSEC_DEFAULT_MM_AUTH_NOT_FOUND:
        Win32ErrorCodeDescription := 'The specified quick mode policy was not found.';
    Win32ErrorCodes.ERROR_IPSEC_DEFAULT_QM_POLICY_NOT_FOUND:
        Win32ErrorCodeDescription := 'The manifest file contains one or more syntax errors.';
    Win32ErrorCodes.ERROR_IPSEC_TUNNEL_FILTER_EXISTS:
        Win32ErrorCodeDescription :=
            'The application attempted to activate a disabled activation context.';
    Win32ErrorCodes.ERROR_IPSEC_TUNNEL_FILTER_NOT_FOUND:
        Win32ErrorCodeDescription :=
            'The requested lookup key was not found in any active activation context.';
    Win32ErrorCodes.ERROR_IPSEC_MM_FILTER_PENDING_DELETION:
        Win32ErrorCodeDescription := 'The Main Mode filter is pending deletion.';
    Win32ErrorCodes.ERROR_IPSEC_TRANSPORT_FILTER_PENDING_DELETION:
        Win32ErrorCodeDescription := 'The transport filter is pending deletion.';
    Win32ErrorCodes.ERROR_IPSEC_TUNNEL_FILTER_PENDING_DELETION:
        Win32ErrorCodeDescription := 'The tunnel filter is pending deletion.';
    Win32ErrorCodes.ERROR_IPSEC_MM_POLICY_PENDING_DELETION:
        Win32ErrorCodeDescription := 'The Main Mode policy is pending deletion.';
    Win32ErrorCodes.ERROR_IPSEC_MM_AUTH_PENDING_DELETION:
        Win32ErrorCodeDescription := 'The Main Mode authentication bundle is pending deletion.';
    Win32ErrorCodes.ERROR_IPSEC_QM_POLICY_PENDING_DELETION:
        Win32ErrorCodeDescription := 'The Quick Mode policy is pending deletion.';
    Win32ErrorCodes.ERROR_IPSEC_IKE_AUTH_FAIL:
        Win32ErrorCodeDescription := 'IKE authentication credentials are unacceptable.';
    Win32ErrorCodes.ERROR_IPSEC_IKE_ATTRIB_FAIL:
        Win32ErrorCodeDescription := 'IKE security attributes are unacceptable.';
    Win32ErrorCodes.ERROR_IPSEC_IKE_NEGOTIATION_PENDING:
        Win32ErrorCodeDescription := 'IKE Negotiation in progress.';
    Win32ErrorCodes.ERROR_IPSEC_IKE_GENERAL_PROCESSING_ERROR:
        Win32ErrorCodeDescription := 'General processing error.';
    Win32ErrorCodes.ERROR_IPSEC_IKE_TIMED_OUT:
        Win32ErrorCodeDescription := 'Negotiation timed out.';
    Win32ErrorCodes.ERROR_IPSEC_IKE_NO_CERT:
        Win32ErrorCodeDescription := 'IKE failed to find valid machine certificate.';
    Win32ErrorCodes.ERROR_IPSEC_IKE_SA_DELETED:
        Win32ErrorCodeDescription := 'IKE SA deleted by peer before establishment completed.';
    Win32ErrorCodes.ERROR_IPSEC_IKE_SA_REAPED:
        Win32ErrorCodeDescription := 'IKE SA deleted before establishment completed.';
    Win32ErrorCodes.ERROR_IPSEC_IKE_MM_ACQUIRE_DROP:
        Win32ErrorCodeDescription := 'Negotiation request sat in Queue too long.';
    Win32ErrorCodes.ERROR_IPSEC_IKE_QM_ACQUIRE_DROP:
        Win32ErrorCodeDescription := 'Negotiation request sat in Queue too long.';
    Win32ErrorCodes.ERROR_IPSEC_IKE_QUEUE_DROP_MM:
        Win32ErrorCodeDescription := 'Negotiation request sat in Queue too long.';
    Win32ErrorCodes.ERROR_IPSEC_IKE_QUEUE_DROP_NO_MM:
        Win32ErrorCodeDescription := 'Negotiation request sat in Queue too long.';
    Win32ErrorCodes.ERROR_IPSEC_IKE_DROP_NO_RESPONSE:
        Win32ErrorCodeDescription := 'No response from peer.';
    Win32ErrorCodes.ERROR_IPSEC_IKE_MM_DELAY_DROP:
        Win32ErrorCodeDescription := 'Negotiation took too long.';
    Win32ErrorCodes.ERROR_IPSEC_IKE_QM_DELAY_DROP:
        Win32ErrorCodeDescription := 'Negotiation took too long.';
    Win32ErrorCodes.ERROR_IPSEC_IKE_ERROR:
        Win32ErrorCodeDescription := 'Unknown error occurred.';
    Win32ErrorCodes.ERROR_IPSEC_IKE_CRL_FAILED:
        Win32ErrorCodeDescription := 'Certificate Revocation Check failed.';
    Win32ErrorCodes.ERROR_IPSEC_IKE_INVALID_KEY_USAGE:
        Win32ErrorCodeDescription := 'Invalid certificate key usage.';
    Win32ErrorCodes.ERROR_IPSEC_IKE_INVALID_CERT_TYPE:
        Win32ErrorCodeDescription := 'Invalid certificate type.';
    Win32ErrorCodes.ERROR_IPSEC_IKE_NO_PRIVATE_KEY:
        Win32ErrorCodeDescription := 'No private key associated with machine certificate.';
    Win32ErrorCodes.ERROR_IPSEC_IKE_DH_FAIL:
        Win32ErrorCodeDescription := 'Failure in Diffie-Helman computation.';
    Win32ErrorCodes.ERROR_IPSEC_IKE_INVALID_HEADER:
        Win32ErrorCodeDescription := 'Invalid header.';
